// TwinCAT 3 PLC project PMS238
// ProgramVersion: 3.1.4023.0
// libraries:
//   Tc2_Math, * (Beckhoff Automation GmbH)
//   Tc2_ModbusSrv, * (Beckhoff Automation GmbH)
//   Tc2_Standard, * (Beckhoff Automation GmbH)
//   Tc2_SUPS, * (Beckhoff Automation GmbH)
//   Tc2_System, * (Beckhoff Automation GmbH)
//   Tc2_Utilities, * (Beckhoff Automation GmbH)
//   Tc3_Module, * (Beckhoff Automation GmbH)
//   Tc3_PMS_Ex, * (Beckhoff Automation GmbH)
// project tree:
//   DUTs/ AliasOnlyThisProject.TcDUT, E_CompareTime.TcDUT
//   DUTs/ION9000/ E_PM_ION9000_Address.TcDUT
//   DUTs/PM_Simulate/ E_listMeterName.TcDUT, E_PM_Simulate.TcDUT
//   Function/ CompareTime.TcPOU, FgenerateRandom.TcPOU, FUN_Compare_Timestructs.TcPOU (not stored), F_RoundLrealEx.TcPOU, IsGoodData.TcPOU, TimeStruct_To_sTimeAveva.TcPOU
//   GVLs/ GVL.TcGVL, pmDev.TcGVL
//   / PersistanceData.TcTTO, PlcTask.TcTTO
//   Persistance/ Prg_Persistance.TcPOU
//   POUs/CalAccum/ FB_CalCulateAccumulation.TcPOU
//   POUs/CrossCheckTime/ FB_TimeCrossCheck2System.TcPOU (not stored)
//   POUs/FIFO/ FB_FIFO_Lreal.TcPOU, FB_FIFO_TimeStruct.TcPOU (not stored), FB_Universal_FIFO.TcPOU, I_FIFO_Lreal.TcIO (not stored), I_FIFO_Timestruct.TcIO (not stored), I_Universal_FIFO.TcIO (not stored)
//   POUs/Metters/ FB_InitPM.TcPOU, FB_PM_ION_9000.TcPOU, FB_ReadPM5350.TcPOU, FB_READPM5500.TcPOU
//   POUs/Platform/File Logger/ FB_FileLogger.TcPOU (not stored), I_FileLogger.TcIO (not stored)
//   POUs/Platform/ PRG_MachineLogger.TcPOU
//   POUs/Program/ IP231.TcPOU, IP232.TcPOU, IP233.TcPOU, IP234.TcPOU, Ip235.TcPOU, IP236.TcPOU, IP237.TcPOU, MAIN.TcPOU, PmReport2.TcPOU
//   TEST/ FB_PmSimulate.TcPOU, PgrTest.TcPOU, PGRTestFB.TcPOU
//   Universal/DUTs/Utilities/File Logger/ E_FileLoggerAddLogsState.TcDUT (not stored), E_FileLoggerInitState.TcDUT (not stored), E_FileLoggerSetNewPathState.TcDUT (not stored), E_FileLoggerState.TcDUT (not stored)
//   Universal/Utilities/StringMerge/ FUN_MergeLongStrings10.TcPOU (not stored), FUN_MergeStrings10.TcPOU (not stored), FUN_MergeStrings3.TcPOU (not stored), FUN_MergeStrings4.TcPOU (not stored), FUN_MergeStrings5.TcPOU (not stored), FUN_MergeStrings6.TcPOU (not stored)
// real-time tasks:
//   TASK PlcTask: cycle T#10ms, priority 20, ADS port 350
//   TASK PersistanceData: cycle T#2ms, priority 2, ADS port 351

CONFIGURATION PMS238
    RESOURCE PLC ON TwinCAT3
        TASK PersistanceData(INTERVAL := T#2ms, PRIORITY := 2);
        TASK PlcTask(INTERVAL := T#10ms, PRIORITY := 20);
        PROGRAM Prg_Persistance WITH PersistanceData : Prg_Persistance;
        PROGRAM MAIN WITH PlcTask : MAIN;
        PROGRAM PRG_MachineLogger WITH PlcTask : PRG_MachineLogger;
        PROGRAM PmReport2 WITH PlcTask : PmReport2;
    END_RESOURCE
END_CONFIGURATION

// ---- DUTs/AliasOnlyThisProject.TcDUT
TYPE AliasOnlyThisProject :
STRUCT 
	systemTime : TIMESTRUCT;
	bValid : BOOL := true;
END_STRUCT
END_TYPE

// ---- DUTs/E_CompareTime.TcDUT
{attribute 'strict'}
TYPE E_CompareTime :
(
	INVALID_PRE_TIME		:= 0,
	NEW_MINUTE := 5,
	NEW_HOUR := 10,
	NEW_DAY	:= 20,
	NEW_MONTH := 30,
	NEW_YEAR	:= 32,
	SAME_MINUTE := 35,
	SAME_HOUR := 40,
	SAME_DAY := 50,
	SAME_MONTH := 60,
	SAME_YEAR  := 70
);
END_TYPE

// ---- DUTs/ION9000/E_PM_ION9000_Address.TcDUT

TYPE E_PM_ION9000_Address :
(
		
		//ION9000_E_Current_Unbalane_A :=    3012  
		//ION9000_E_Current_Unbalane_B :=    3014  
		//ION9000_E_Current_Unbalane_C :=    3016  
		ION9000_E_Current_Unbalane_Worst :=    3018,  
		//ION9000_E_Current_Unbalane_AB :=    3038  
		//ION9000_E_Current_Unbalane_BC :=    3040  
		//ION9000_E_Current_Unbalane_CA :=    3042  
		//ION9000_E_Current_Unbalane_LL_Worst :=    3044  
		//ION9000_E_Current_Unbalane_AN :=    3046  
		//ION9000_E_Current_Unbalane_BN :=    3048  
		//ION9000_E_Current_Unbalane_CN :=    3050  
		//ION9000_E_Current_Unbalane_LN_Worst:= ,
		ION9000_E_Voltage_Unbalane_LN_Worst :=    3052,  
		ION9000_E_Real_PowerA :=    3054  ,
		ION9000_E_Real_PowerB :=    3056  ,
		ION9000_E_Real_PowerC :=    3058  ,
		ION9000_E_Real_PowerTotal :=    3060  ,
		ION9000_E_Reactive_PowerA :=    3062  ,
		ION9000_E_Reactive_PowerB :=    3064  ,
		ION9000_E_Reactive_PowerC :=    3066  ,
		ION9000_E_Reactive_PowerTotal :=    3068 , 
		ION9000_E_Apparent_PowerA :=    3070  ,
		ION9000_E_Apparent_PowerB :=    3072  ,
		ION9000_E_Apparent_PowerC :=    3074  ,
		ION9000_E_Apparent_PowerTotal :=    3076  ,
		ION9000_E_Voltage_AB :=    3020 , 
		ION9000_E_Voltage_BC :=    3022  ,
		ION9000_E_Voltage_CA :=    3024  ,
		ION9000_E_Voltage_LLAvg :=    3026  ,
		ION9000_E_Voltage_AN :=    3028  ,
		ION9000_E_Voltage_BN :=    3030  ,
		ION9000_E_Voltage_CN :=    3032  ,
		ION9000_E_Voltage_NG	:= 3034,
		ION9000_E_Voltage_LNAvg :=    3036  ,
//		ION9000_E_THDF_Voltage_AB :=    22  ,
//		ION9000_E_THDF_Voltage_BC :=    24  ,
//		ION9000_E_THDF_Voltage_CA :=    26  ,
		//ION9000_E_THDF_Voltage_LL :=    28  ,
		ION9000_E_THDF_Voltage_AN :=    21330, 
		ION9000_E_THDF_Voltage_BN :=    21332, 
		ION9000_E_THDF_Voltage_CN :=    21334, 
		ION9000_E_THDF_Voltage_LN :=    21336,  
//		ION9000_E_thdR_Voltage_AB :=    40,  
//		ION9000_E_thdR_Voltage_BC :=    42,  
//		ION9000_E_thdR_Voltage_CA :=    44 , 
//		ION9000_E_thdR_Voltage_LL :=    45 , 
//		ION9000_E_thdR_Voltage_AN :=    48 , 
//		ION9000_E_thdR_Voltage_BN :=    50 , 
//		ION9000_E_thdR_Voltage_CN :=    52 , 
//		ION9000_E_thdR_Voltage_LN :=    56 , 
		ION9000_E_Current_A :=    3000 , 
		ION9000_E_Current_B :=    3002,  
		ION9000_E_Current_C :=    3004  ,
		ION9000_E_Current_N :=    3006 , 
		ION9000_E_Current_G :=    3008  ,
		ION9000_E_Current_Avg :=    3010 , 
		ION9000_E_THDF_Current_A :=    21300 , 
		ION9000_E_THDF_Current_B :=  	21302, 
		ION9000_E_THDF_Current_C :=   21304  ,
		ION9000_E_THDF_Current_N :=    21306, 
		ION9000_E_THDF_Current_G :=   21308  ,
//		ION9000_E_thdR_Current_A :=    10  ,
//		ION9000_E_thdR_Current_B :=    12  ,
//		ION9000_E_thdR_Current_C :=    14  ,
//		ION9000_E_thdR_Current_N :=    16  ,
//		ION9000_E_thdR_Current_G :=    18  ,
//		ION9000_E_Total_Demand_Distortion :=    20  
		ION9000_E_RealEnergy_IntoLoad :=    3204  ,
		ION9000_E_RealEnergy_OutLoad :=    3208 , 
		ION9000_E_RealEnergy_Absolute :=    3212  ,
		ION9000_E_RealEnergy_Signed :=    3216  ,
		ION9000_E_ReactiveEnergy_IntoLoad :=    3220 , 
		ION9000_E_ReactiveEnergy_OutLoad :=    3224  ,
		ION9000_E_ReactiveEnergy_Absolute :=    3228  ,
		ION9000_E_ReactiveEnergy_Signed :=    3232  ,
		ION9000_E_ApparentEnergy_IntoLoad :=    3236  ,
		ION9000_E_ApparentEnergy_OutLoad :=    3240  ,
		ION9000_E_ApparentEnergy :=    3244  ,
		ION9000_E_ApparentEnergy_Delivered_Received :=    3248  ,
		ION9000_E_Frequency :=    3110  ,
		ION9000_E_PowerFactor :=    3150
	
);
END_TYPE

// ---- DUTs/PM_Simulate/E_listMeterName.TcDUT
{attribute 'strict'}
TYPE E_listMeterName :
(
	LV01  := 0,
	DB_PR1_1  := 1,
	DB1  := 2,
	DB2  := 3,
	DB3  := 4,
	DB4  := 5,
	DB1_1  := 6,
	DB2_1  := 7,
	DB3_1  := 8,
	DB4_1  := 9,
	DB5  := 10,
	DB6  := 11,
	DB7  := 12,
	DB_MR  := 13,
	DB5_1  := 14,
	DB6_1  := 15,
	DB7_1  := 16,
	LV02  := 17,
	DB_PR1_2  := 18,
	DB_AIRCOMP  := 19,
	DB_AHU  := 20,
	DB8  := 21,
	DB9  := 22,
	DB10  := 23,
	DB8_1  := 24,
	DB9_1  := 25,
	DB10_1  := 26,
	A1  := 27,
	A2  := 28,
	A3  := 29,
	A4  := 30,
	A5  := 31,
	LP_PR1A  := 32,
	LP_PR1B  := 33,
	LP_PR2A  := 34,
	LP_PR2B  := 35,
	LP_PR3A  := 36,
	DB_WH  := 37,
	LP_PR3B  := 38,
	LP_PR4A  := 39,
	LP_PR4B  := 40,
	LP_BM  := 41,
	DB_BM  := 42,
	LV03  := 43,
	DB_MVAC1  := 44,
	DB_MVAC2  := 45,
	DB_OFF2  := 46,
	LP_EL1  := 47,
	LP_EL2  := 48,
	DB_OFF1  := 49,
	DB_KIT  := 50,
	LP_WH2  := 51,
	LP_WH1  := 52,
	CH4  := 53,
	CH5  := 54,
	CH6  := 55,
	LV04  := 56,
	DB_PR2  := 57,
	DB11  := 58,
	DB12  := 59,
	DB13  := 60,
	DB14  := 61,
	DB11_1  := 62,
	DB12_1  := 63,
	DB13_1  := 64,
	DB14_1  := 65,
	DB15  := 66,
	DB15_1  := 67,
	LP_PR5A  := 68,
	LP_PR5B  := 69,
	LP_PR6A  := 70,
	LP_PR6B  := 71,
	 DB1_2	 :=72,
	 DB2_2	 :=73,
	 DB3_2	 :=74,
	 DB4_2	 :=75,
	 DB5_2	 :=76,
	 DB6_2	 :=77,
	 DB7_2	 :=78,
	 DB8_2	 :=79,
	 DB9_2	 :=80,
	 DB10_2	 :=81,
	 DB11_2	 :=82,
	 DB12_2	 :=83,
	 DB13_2	 :=84,
	 DB14_2	 :=85,
	 DB15_2	 :=86
);
END_TYPE

// ---- DUTs/PM_Simulate/E_PM_Simulate.TcDUT

{attribute 'strict'}
TYPE E_PM_Simulate :
(
	
	PM_SIMU_WAIT := 0,
	PM_SIMU_UPDATE := 10,
	PM_SIMU_READ_FAULT := 20
);
END_TYPE

// ---- GVLs/GVL.TcGVL

VAR_GLOBAL
	fbMachineLogger : FB_FileLogger;
	fbMachineTime	: AliasOnlyThisProject;
END_VAR
VAR_GLOBAL CONSTANT
	TIME_INIT	: TIME := T#30S;
END_VAR

// ---- GVLs/pmDev.TcGVL
{attribute 'qualified_only'}
VAR_GLOBAL
	DB01_02_5350		: ST_PowerMeter; //DB12.1
	DB01_03_5350		: ST_PowerMeter; //DB11.1
	DB01_05_5350		: ST_PowerMeter; //LP-PR6B
	DB01_06_5350		: ST_PowerMeter; //LP-PR6A
	DB01_12_5350		: ST_PowerMeter; //LP-WH2
	
	DB01_01_5500		: ST_PowerMeter; //DB12
	DB01_04_5500		: ST_PowerMeter; //DB11
	DB01_07_5500		: ST_PowerMeter; //DB-PR2
	DB01_11_5500		: ST_PowerMeter; //LP-WH1
	DB01_18_5500		: ST_PowerMeter; //DB-WH
	DB01_20_5500		: ST_PowerMeter; //LP-BM
	DB01_22_5500		: ST_PowerMeter; //DB-BM 
	
	DB02_01_5350		: ST_PowerMeter; //DB13.1
	DB02_03_5350		: ST_PowerMeter; //DB15.1
	DB02_05_5350		: ST_PowerMeter; //DB14.1 
	DB02_07_5350		: ST_PowerMeter; //LP-PR5B
	DB02_08_5350		: ST_PowerMeter; //LP-PR5A
	
	DB02_02_5500		: ST_PowerMeter; //DB13
	DB02_04_5500		: ST_PowerMeter; //DB15
	DB02_06_5500		: ST_PowerMeter; //DB14
	
	
	DB03_01_5350		: ST_PowerMeter; //DB7.1
	DB03_03_5350		: ST_PowerMeter; //DB5.1 
	DB03_05_5350		: ST_PowerMeter; //DB6.1
	DB03_07_5350		: ST_PowerMeter; //LP-PR3B
	DB03_08_5350		: ST_PowerMeter; //LP-PR3A
	
	DB03_02_5500		: ST_PowerMeter; //DB7
	DB03_04_5500		: ST_PowerMeter; //DB5
	DB03_06_5500		: ST_PowerMeter; //DB6
	
	DB04_01_5350		: ST_PowerMeter; //DB4.1 
	DB04_03_5350		: ST_PowerMeter; //DB3.1 
	DB04_05_5350		: ST_PowerMeter; //DB2.1 
	DB04_07_5350		: ST_PowerMeter; //LP-PR4B
	DB04_08_5350		: ST_PowerMeter; //LP-PR4A
	
	DB04_02_5500		: ST_PowerMeter; //DB4
	DB04_04_5500		: ST_PowerMeter; //DB3
	DB04_06_5500		: ST_PowerMeter; //DB2
	
	
	DB05_01_5350		: ST_PowerMeter; //LP-PR1A
	DB05_02_5350		: ST_PowerMeter; //LP-PR1B
	DB05_03_5350		: ST_PowerMeter; //DB8.1 
	DB05_05_5350		: ST_PowerMeter; //DB9.1 
	DB05_07_5350		: ST_PowerMeter; //DB10.1
	DB05_09_5350		: ST_PowerMeter; //DB1.1
	DB05_21_5350		: ST_PowerMeter; //LP-PR2B
	DB05_22_5350		: ST_PowerMeter; //LP-PR2A
	
	DB05_04_5500		: ST_PowerMeter; //DB8
	DB05_06_5500		: ST_PowerMeter; //DB9
	DB05_08_5500		: ST_PowerMeter; //DB10
	DB05_10_5500		: ST_PowerMeter; //DB1 
	
	DB06_01_5500		: ST_PowerMeter; //LP-EL2
	DB06_02_5500		: ST_PowerMeter; //LV-SECTION4
	DB06_03_5500		: ST_PowerMeter; //LP-EL1
	DB06_04_5500		: ST_PowerMeter; //LV-SECTION3
	DB06_05_5500		: ST_PowerMeter; //DB-PR1 (S2) 
	DB06_06_5500		: ST_PowerMeter; //DB-PR1(S1)
	DB06_07_5500		: ST_PowerMeter; //DB-AHU
	DB06_08_5500		: ST_PowerMeter; //DB-OFF1
	DB06_11_5500		: ST_PowerMeter; //DB-MR
	DB06_33_5500		: ST_PowerMeter; //DB-KIT
	DB06_38_5500		: ST_PowerMeter; //DB-OFF2
	
	DB07_01_5500		: ST_PowerMeter; //LV-SECTION1
	DB07_02_5500		: ST_PowerMeter; // LV-SECTION2
	DB07_03_5500		: ST_PowerMeter; //DB-AIRCOMP 
	DB07_04_5500		: ST_PowerMeter; //DB-MVAC2
	DB07_05_5500		: ST_PowerMeter; //DB-MVAC1
	///////////////////////////////////////////////Sun update Code
	DB07_06_5350		: ST_PowerMeter; // A1
	DB07_07_5350		: ST_PowerMeter; //A2
	DB07_08_5350		: ST_PowerMeter; //A3
	DB07_09_5350		: ST_PowerMeter; //A4
	DB07_10_5350		: ST_PowerMeter; //A5
	DB07_11_5350		: ST_PowerMeter; //CH4
	DB07_12_5350		: ST_PowerMeter; //CH5
	DB07_13_5350		: ST_PowerMeter; //CH6
	/////// virtual metter 
	PowerMeter_Db1_2	: st_powerMeter;// DB1.2
	PowerMeter_Db2_2	: ST_PowerMeter;
	PowerMeter_db3_2	: ST_PowerMeter;
	PowerMeter_db4_2	: ST_PowerMeter;
	PowerMeter_db5_2	: ST_PowerMeter;
	powerMeter_db6_2	: ST_PowerMeter;
	PowerMeter_db7_2	: ST_PowerMeter;
	PowerMeter_db8_2	: ST_PowerMeter;
	PowerMeter_db9_2	: ST_PowerMeter;
	PowerMeter_db10_2	: ST_PowerMeter;
	PowerMeter_db11_2	: ST_PowerMeter;
	PowerMeter_db12_2	: ST_PowerMeter;
	PowerMeter_db13_2	: ST_PowerMeter;
	PowerMeter_db14_2	: ST_PowerMeter;
	PowerMeter_db15_2	: ST_PowerMeter;

	// new meter
	PowerMeter_Lv01		: ST_PowerMeter;
	PowerMeter_Lv02		: ST_PowerMeter;
	PowerMeter_Lv03		: ST_PowerMeter;
	PowerMeter_Lv04		: ST_PowerMeter;

	NT_GetTime : NT_GetTime;
	AvevaTimeStruct : TIMESTRUCT;
	bAlarmDifferentTime2System : BOOL;
END_VAR
VAR_GLOBAL CONSTANT
	TIMESTRUCT_DEFAULT : TIMESTRUCT;
	InvalidValueEnergyIntoload   : LREAL := 1E12; // if Energy Intoload bigger this parameter or lower than (-NanEnergyIntoload) , EnergyIntoload can't be use
	numAllMeter	 :UINT := 87;
	SecondDifferentAllow : UDINT := 300;
END_VAR
// commissioning
VAR_GLOBAL
	bTrigReadCOmmision : BOOL;
END_VAR

// ---- Persistance/Prg_Persistance.TcPOU
PROGRAM Prg_Persistance
VAR
FB_S_UPS_CX8190	: FB_S_UPS_CX81xx;

END_VAR

FB_S_UPS_CX8190(	sNetID :='',
					iPLCPort        := 851, (* PLC Runtime System for writing persistent data *)
  					tTimeout        := DEFAULT_ADS_TIMEOUT, (* ADS Timeout *)
    				eUpsMode        := eSUPS_WrPersistData_Shutdown, (* UPS mode (w/wo writing persistent data, w/wo NO shutdown) *)
   					ePersistentMode := SPDM_2PASS, (* mode for writing persistent data *)
    				tRecoverTime    := T#10S, (* ON time to recover from short power failure in mode eSUPS_WrPersistData_NoShutdown/eSUPS_CheckPowerStatus *)
					);

END_PROGRAM

// ---- POUs/Program/MAIN.TcPOU
PROGRAM MAIN
VAR
	fb_timeCrossCheck	: FB_TimeCrossCheck2System;
	eEgxRead	: UINT := WAIT_EGX_FREE;
END_VAR

VAR CONSTANT
	WAIT_EGX_FREE	: UINT := 0;
	EGX_231 : UINT := 231;
	EGX_232 : UINT := 232;
	EGX_233 : UINT := 233;
	EGX_234 : UINT := 234;
	EGX_235 : UINT := 235;
	EGX_236 : UINT := 236;
	EGX_237 : UINT := 237;
END_VAR

IF FUN_Compare_Timestructs(
	ts1 := pmDev.AvevaTimeStruct, 
	ts2 := pmDev.TIMESTRUCT_DEFAULT
	) = 0 // equal
THEN
	 pmDev.bAlarmDifferentTime2System := FALSE;
	 
ELSE 
	fb_timeCrossCheck(	TimeStruct_Sys1 := pmDev.AvevaTimeStruct,
					TimeStruct_Sys2 := pmDev.NT_GetTime.TIMESTR,
					secondDifferentAllow := pmdev.SecondDifferentAllow,
					bErrorTimeTwoSystem => pmDev.bAlarmDifferentTime2System);
END_IF

pmdev.NT_GetTime(START := FALSE);
pmdev.NT_GetTime(
	START := TRUE,
	TIMESTR => GVL.fbMachineTime.systemTime
); 
					
IP231();
IP232();
IP233();
IP234();
IP235();
IP236();
IP237();
CASE eEgxRead OF
	WAIT_EGX_FREE :
		IF NOT IP231.Busy
		AND NOT IP232.Busy
		AND NOT IP233.Busy
		AND NOT IP234.Busy
		AND NOT IP235.Busy
		AND NOT IP236.Busy
		AND NOT IP237.Busy
		THEN
			eEgxRead := EGX_231;
		END_IF
		
	EGX_231 :
		IP231.Mr_Read();
		IF NOT IP231.Busy THEN
			eEgxRead := EGX_232;
		END_IF
		
	EGX_232 :
		IP232.Mr_Read();
		IF NOT IP232.Busy THEN
			eEgxRead := EGX_233;
		END_IF
		
	EGX_233 :
		IP233.Mr_Read();
		IF NOT IP233.Busy THEN
			eEgxRead := EGX_234;
		END_IF
		
	EGX_234 :
		IP234.Mr_Read();
		IF NOT IP234.Busy THEN
			eEgxRead := EGX_235;
		END_IF
		
	EGX_235 :
		IP235.Mr_Read();
		IF NOT IP235.Busy THEN
			eEgxRead := EGX_236;
		END_IF
		
	EGX_236 :
		IP236.Mr_Read();
		IF NOT IP236.Busy THEN
			eEgxRead := EGX_237;
		END_IF
		
	EGX_237 :
		IP237.Mr_Read();
		IF NOT IP237.Busy THEN
			eEgxRead := WAIT_EGX_FREE;
		END_IF
END_CASE

pmdev.bTrigReadCOmmision := FALSE;
CalculateVirtualMeter(	MeterMain := pmDev.DB05_10_5500 ,
						MeterSub := pmDev.DB05_09_5350,
						MeterVirtual := pmDev.PowerMeter_Db1_2);
						
 CalculateVirtualMeter( MeterMain := pmDev.DB04_06_5500,
                      MeterSub := pmDev.DB04_05_5350,
                       MeterVirtual :=  pmDev.PowerMeter_Db2_2);
 
 CalculateVirtualMeter( MeterMain := pmDev.DB04_04_5500,
                      MeterSub :=  pmDev.DB04_03_5350,
                       MeterVirtual :=  pmDev.PowerMeter_db3_2);
 
 CalculateVirtualMeter( MeterMain := pmDev.DB04_02_5500,
                      MeterSub := pmDev.DB04_01_5350,
                       MeterVirtual :=  pmDev.PowerMeter_db4_2);
 
 CalculateVirtualMeter( MeterMain := pmDev.DB03_04_5500,
                      MeterSub := pmDev.DB03_03_5350,
                       MeterVirtual :=  pmDev.PowerMeter_db5_2);
 
 CalculateVirtualMeter( MeterMain := pmDev.DB03_06_5500,
                      MeterSub := pmDev.DB03_05_5350,
                       MeterVirtual :=  pmDev.powerMeter_db6_2);
 
 CalculateVirtualMeter( MeterMain := pmDev.DB03_02_5500,
                      MeterSub := pmDev.DB03_01_5350,
                       MeterVirtual :=  pmDev.PowerMeter_db7_2);
 
 CalculateVirtualMeter( MeterMain := pmDev.DB05_04_5500,
                      MeterSub := pmDev.DB05_03_5350,
                       MeterVirtual :=  pmDev.PowerMeter_db8_2);
 
 CalculateVirtualMeter( MeterMain := pmDev.DB05_06_5500,
                      MeterSub := pmDev.DB05_05_5350,
                       MeterVirtual :=  pmDev.PowerMeter_db9_2);
 
 CalculateVirtualMeter( MeterMain := pmDev.DB05_08_5500,
                      MeterSub := pmDev.DB05_07_5350,
                       MeterVirtual :=  pmDev.PowerMeter_db10_2);
 
 CalculateVirtualMeter( MeterMain := pmDev.DB01_04_5500,
                      MeterSub := pmDev.DB01_03_5350,
                       MeterVirtual :=  pmDev.PowerMeter_db11_2);
 
 CalculateVirtualMeter( MeterMain :=  pmDev.DB01_01_5500,
                      MeterSub := pmDev.DB01_02_5350,
                       MeterVirtual :=  pmDev.PowerMeter_db12_2);
 
 CalculateVirtualMeter( MeterMain := pmDev.DB02_02_5500,
                      MeterSub := pmDev.DB02_01_5350,
                       MeterVirtual :=  pmDev.PowerMeter_db13_2);
 
 CalculateVirtualMeter( MeterMain := pmDev.DB02_06_5500,
                      MeterSub := pmDev.DB02_05_5350,
                       MeterVirtual :=  pmDev.PowerMeter_db14_2);
 
 CalculateVirtualMeter( MeterMain := pmDev.DB02_04_5500,
                      MeterSub := pmDev.DB02_03_5350,
                       MeterVirtual :=  pmDev.PowerMeter_db15_2);

METHOD CalculateVirtualMeter : BOOL
VAR_INPUT
	MeterMain	: REFERENCE TO  ST_PowerMeter;// meterVirtual := MeterMain - MeterSub
	MeterSub	: REFERENCE TO ST_PowerMeter;// meterVirtual := MeterMain - MeterSub
	MeterVirtual : REFERENCE TO ST_PowerMeter; // meterVirtual := MeterMain - MeterSub
END_VAR
VAR_OUTPUT
	
END_VAR
	MeterVirtual.Basic.Current_Avg := MeterMain.Basic.Current_Avg - MeterSub.Basic.Current_Avg;
	MeterVirtual.Basic.Real_PowerTotal := MeterMain.Basic.Real_PowerTotal - MeterSub.Basic.Real_PowerTotal;
	MeterVirtual.Basic.RealEnergy_IntoLoad  := MeterMain.Basic.RealEnergy_IntoLoad - MeterSub.Basic.RealEnergy_IntoLoad;
END_METHOD

END_PROGRAM

// ---- POUs/Program/IP231.TcPOU
PROGRAM IP231
VAR
	timer				: TON;
	nState				: INT := STATE_INIT;
	
	fbInit231_02_5350			: FB_InitPM;
	fbInit231_03_5350			: FB_InitPM;
	fbInit231_05_5350			: FB_InitPM;
	fbInit231_06_5350			: FB_InitPM;
	fbInit231_12_5350			: FB_InitPM;
	
	fbRead231_02_5350			: FB_ReadPM5350;
	fbRead231_03_5350			: FB_ReadPM5350;
	fbRead231_05_5350			: FB_ReadPM5350;
	fbRead231_06_5350			: FB_ReadPM5350;
	fbRead231_12_5350			: FB_ReadPM5350;
	
	fbInit231_01_5500			: FB_InitPM;
	fbInit231_04_5500			: FB_InitPM;
	fbInit231_07_5500			: FB_InitPM;
	fbInit231_11_5500			: FB_InitPM;
	fbInit231_18_5500			: FB_InitPM;
	fbInit231_20_5500			: FB_InitPM;
	fbInit231_22_5500			: FB_InitPM;
	
	fbRead231_01_5500			: FB_ReadPM5500;
	fbRead231_04_5500			: FB_ReadPM5500;
	fbRead231_07_5500			: FB_ReadPM5500;
	
	//Update 29-8-2022
	fbRead231_11_5500			: FB_ReadPM5350;
	
	fbRead231_18_5500			: FB_ReadPM5500;
	fbRead231_20_5500			: FB_ReadPM5500;
	fbRead231_22_5500			: FB_ReadPM5500;
END_VAR

VAR CONSTANT
	STATE_INIT			:	INT		:= 0;
	STATE_WAIT_CMD		: 	INT		:= 5;
	STATE_READ2			:	INT		:= 20;
	STATE_READ3			:	INT		:= 30;
	STATE_READ5			:	INT		:= 50;
	STATE_READ6			:	INT		:= 60;
	STATE_READ12		:	INT		:= 90;
	STATE_READ1			:	INT		:= 10;
	STATE_READ4			:	INT		:= 40;
	STATE_READ7			:	INT		:= 70;
	STATE_READ11		:	INT		:= 110;
	STATE_READ18		:	INT		:= 180;
	STATE_READ20		:	INT		:= 200;
	STATE_READ22		:	INT		:= 220;
END_VAR

CASE nState OF
	STATE_INIT:
		fbInit231_02_5350(	sIpAddress	:= '10.91.37.231',
							nPort		:= 502,
							nUnitID		:= 2,
							PM			:= pmDev.DB01_02_5350);
		fbInit231_03_5350(	sIpAddress	:= '10.91.37.231',
							nPort		:= 502,
							nUnitID		:= 03,
							PM			:= pmDev.DB01_03_5350);
		fbInit231_05_5350(	sIpAddress	:= '10.91.37.231',
							nPort		:= 502,
							nUnitID		:= 5,
							PM			:= pmDev.DB01_05_5350);
		fbInit231_06_5350(	sIpAddress	:= '10.91.37.231',
							nPort		:= 502,
							nUnitID		:= 6,
							PM			:= pmDev.DB01_06_5350);
							
		fbInit231_11_5500(	sIpAddress	:= '10.91.37.231',
							nPort		:= 502,
							nUnitID		:= 11,
							PM			:= pmDev.DB01_11_5500);
							
		fbInit231_12_5350(	sIpAddress	:= '10.91.37.231',
							nPort		:= 502,
							nUnitID		:= 12,
							PM			:= pmDev.DB01_12_5350);
							
		fbInit231_01_5500(	sIpAddress	:= '10.91.37.231',
							nPort		:= 502,
							nUnitID		:= 1,
							PM			:= pmDev.DB01_01_5500);
		fbInit231_04_5500(	sIpAddress	:= '10.91.37.231',
							nPort		:= 502,
							nUnitID		:= 4,
							PM			:= pmDev.DB01_04_5500);
		fbInit231_07_5500(	sIpAddress	:= '10.91.37.231',
							nPort		:= 502,
							nUnitID		:= 7,
							PM			:= pmDev.DB01_07_5500);
		
		fbInit231_18_5500(	sIpAddress	:= '10.91.37.231',
							nPort		:= 502,
							nUnitID		:= 18,
							PM			:= pmDev.DB01_18_5500);
		fbInit231_20_5500(	sIpAddress	:= '10.91.37.231',
							nPort		:= 502,
							nUnitID		:= 20,
							PM			:= pmDev.DB01_20_5500);
		fbInit231_22_5500(	sIpAddress	:= '10.91.37.231',
							nPort		:= 502,
							nUnitID		:= 22,
							PM			:= pmDev.DB01_22_5500);
							
		timer(In:=TRUE, PT:= TIME_INIT);
		IF timer.Q THEN
			timer(In := FALSE);
			nState	:= STATE_WAIT_CMD;
		END_IF
	STATE_WAIT_CMD:
		;
	STATE_READ2:
		fbRead231_02_5350(
			bExecute:=TRUE,
			PM:= pmDev.DB01_02_5350);
		IF NOT fbRead231_02_5350.Q THEN
			nState	:= STATE_READ3;
			fbRead231_02_5350(
				bExecute:=FALSE,
				PM:= pmDev.DB01_02_5350);
		END_IF
		
	STATE_READ3:
		fbRead231_03_5350(
			bExecute:=TRUE,
			PM:= pmDev.DB01_03_5350);
		IF NOT fbRead231_03_5350.Q THEN
			nState	:= STATE_READ5;
			fbRead231_03_5350(
				bExecute:=FALSE,
				PM:= pmDev.DB01_03_5350);
		END_IF	
	
	STATE_READ5:
		fbRead231_05_5350(
			bExecute:=TRUE,
			PM:= pmDev.DB01_05_5350);
		IF NOT fbRead231_05_5350.Q THEN
			nState	:= STATE_READ6;
			fbRead231_05_5350(
				bExecute:=FALSE,
				PM:= pmDev.DB01_05_5350);
		END_IF	
		
	STATE_READ6:
		fbRead231_06_5350(
			bExecute:=TRUE,
			PM:= pmDev.DB01_06_5350);
		IF NOT fbRead231_06_5350.Q THEN
			nState	:= STATE_READ11;
			fbRead231_06_5350(
			bExecute:=FALSE,
			PM := pmDev.DB01_06_5350);
		END_IF
		
	STATE_READ11:
	
		
		fbRead231_11_5500(
			bExecute:=TRUE,
			PM:= pmDev.DB01_11_5500);
		IF NOT fbRead231_11_5500.Q THEN
			nState	:= STATE_READ12;
			fbRead231_11_5500(
				bExecute:=FALSE,
				PM:= pmDev.DB01_11_5500);
		END_IF
		
	STATE_READ12:
		fbRead231_12_5350(
			bExecute:=TRUE,
			PM:= pmDev.DB01_12_5350);
		IF NOT fbRead231_12_5350.Q THEN
			nState	:= STATE_READ1;
			fbRead231_12_5350(
				bExecute:=FALSE,
				PM:= pmDev.DB01_12_5350);
		END_IF	
	STATE_READ1:
		fbRead231_01_5500(
			bExecute:=TRUE,
			PM:= pmDev.DB01_01_5500);
		IF NOT fbRead231_01_5500.Q THEN
			nState	:= STATE_READ4;
			fbRead231_01_5500(
				bExecute:=FALSE,
				PM:= pmDev.DB01_01_5500);
		END_IF
	STATE_READ4:
		fbRead231_04_5500(
			bExecute:=TRUE,
			PM:= pmDev.DB01_04_5500);
		IF NOT fbRead231_04_5500.Q THEN
			nState	:= STATE_READ7;
			fbRead231_04_5500(
				bExecute:=FALSE,
				PM:= pmDev.DB01_04_5500);
		END_IF
	
	STATE_READ7:
		fbRead231_07_5500(
			bExecute:=TRUE,
			PM:= pmDev.DB01_07_5500);
		IF NOT fbRead231_07_5500.Q THEN
			nState	:= STATE_READ18;
			fbRead231_07_5500(
				bExecute:=FALSE,
				PM:= pmDev.DB01_07_5500);
		END_IF
		
	STATE_READ18:
		fbRead231_18_5500(
			bExecute:=TRUE,
			PM:= pmDev.DB01_18_5500);
		IF NOT fbRead231_18_5500.Q THEN
			nState	:= STATE_READ20;
			fbRead231_18_5500(
				bExecute:=FALSE,
				PM:= pmDev.DB01_18_5500);
		END_IF
		
	STATE_READ20:
		fbRead231_20_5500(
			bExecute:=TRUE,
			PM:= pmDev.DB01_20_5500);
		IF NOT fbRead231_20_5500.Q THEN
			nState	:= STATE_READ22;
			fbRead231_20_5500(
				bExecute:=FALSE,
				PM:= pmDev.DB01_20_5500);
		END_IF
	
	STATE_READ22:
		fbRead231_22_5500(
			bExecute:=TRUE,
			PM:= pmDev.DB01_22_5500);
		IF NOT fbRead231_22_5500.Q THEN
			nState	:= STATE_WAIT_CMD;
			fbRead231_22_5500(
				bExecute:=FALSE,
				PM:= pmDev.DB01_22_5500);
		END_IF
	
END_CASE

PROPERTY Busy : Bool
GET
Busy := nState <> STATE_WAIT_CMD;
END_GET
END_PROPERTY

METHOD Mr_Read : BOOL
VAR_INPUT
END_VAR
IF nState = STATE_WAIT_CMD THEN
	nState := STATE_READ2;
END_IF
END_METHOD

END_PROGRAM

// ---- POUs/Metters/FB_InitPM.TcPOU
FUNCTION_BLOCK FB_InitPM
VAR_INPUT
	sIpAddress		: STRING;
	nUnitID			: BYTE;
	nPort			: UINT;
END_VAR

VAR_OUTPUT
END_VAR

VAR_IN_OUT
	PM		:	ST_PowerMeter;
END_VAR

VAR
END_VAR

(******** Init Connection **************)
PM.Conn.sIPAddress		:= sIpAddress;
PM.Conn.nUnitID			:= nUnitID;
PM.Conn.nPort			:= nPort;

END_FUNCTION_BLOCK

// ---- POUs/Metters/FB_ReadPM5350.TcPOU
FUNCTION_BLOCK FB_ReadPM5350 EXTENDS ReadPm5350

VAR_OUTPUT
END_VAR
VAR PERSISTENT
	validEnvergyIntoLoad : LREAL;
END_VAR
(*VAR_IN_OUT
	PM		:	ST_PowerMeter;
END_VAR*)
VAR
	bOtherDataGood : BOOL;
END_VAR

SUPER^(PM:= THIS^.PM,
		bExecute := bExecute);

bOtherdataGood := 	IsGoodData( pm.Basic.Voltage_LLAvg )
				AND IsGoodData( pm.Basic.Current_Avg)
				AND IsGoodData(	pm.Basic.Frequency)
				AND IsGoodData( pm.Basic.Voltage_AN)
				AND IsGoodData(	pm.Basic.Voltage_AB)
				AND IsGoodData( pm.Basic.Voltage_BN)
				AND IsGoodData(	pm.Basic.Voltage_BC)
				AND IsGoodData( pm.Basic.Voltage_CN)
				AND IsGoodData(	pm.Basic.Voltage_CA);
				
				
IF IsGoodData (pm.Basic.RealEnergy_IntoLoad ) AND bOtherDataGood THEN
	;// pm.Basic.RealEnergy_IntoLoad still it
	validEnvergyIntoLoad := pm.Basic.RealEnergy_IntoLoad;
ELSE
	pm.Basic.RealEnergy_IntoLoad := validEnvergyIntoLoad;
END_IF

//round value
	(*PM.Basic.RealEnergy_IntoLoad := F_RoundLrealEx(	lrIn 	:= PM.Basic.RealEnergy_IntoLoad,
										iPrecision 	:= 0);*)
												
	PM.Basic.PowerFactor := F_RoundLrealEx(	lrIn 	:= PM.Basic.PowerFactor,
								iPrecision 	:= 2);

END_FUNCTION_BLOCK

// ---- Function/IsGoodData.TcPOU
FUNCTION IsGoodData : BOOL// check into load data not nan and too big or too low
VAR_INPUT
	dataLr : LREAL;
END_VAR
VAR
END_VAR

IF LrealIsNaN( dataLr ) THEN
	IsGoodData := FALSE;
ELSIF dataLr > pmDev.InvalidValueEnergyIntoload OR dataLr <  0.0001 THEN
	IsGoodData := FALSE;
ELSE
	IsGoodData := True;
END_IF

END_FUNCTION

// ---- Function/F_RoundLrealEx.TcPOU
FUNCTION F_RoundLrealEx : LREAL
VAR_INPUT
	lrIn : LREAL;
	iPrecision : UINT;
END_VAR
VAR
	lrTemp	: LREAL;
END_VAR

lrTemp := lrIn * EXPT(10,iPrecision);
lrTemp := LTRUNC(lrTemp);
F_RoundLrealEx := lrTemp / EXPT(10,iPrecision);

END_FUNCTION

// ---- POUs/Metters/FB_READPM5500.TcPOU
FUNCTION_BLOCK FB_READPM5500 EXTENDS ReadPm5500

VAR_OUTPUT
END_VAR
VAR PERSISTENT 
	validEnvergyIntoLoad : LREAL;
END_VAR
(*VAR_IN_OUT
	PM		:	ST_PowerMeter;
END_VAR*)
VAR
	bOtherDataGood : BOOL;
END_VAR

SUPER^(PM:= THIS^.PM,
		bExecute := bExecute);

bOtherdataGood := 	IsGoodData( pm.Basic.Voltage_LLAvg )
				AND IsGoodData ( pm.Basic.Current_Avg)
				AND IsGoodData(	pm.Basic.Frequency)
				AND IsGoodData( pm.Basic.Voltage_AN)
				AND IsGoodData(	pm.Basic.Voltage_AB)
				AND IsGoodData( pm.Basic.Voltage_BN)
				AND IsGoodData(	pm.Basic.Voltage_BC)
				AND IsGoodData( pm.Basic.Voltage_CN)
				AND IsGoodData(	pm.Basic.Voltage_CA);

				
IF IsGoodData (pm.Basic.RealEnergy_IntoLoad ) AND bOtherDataGood THEN
	;// pm.Basic.RealEnergy_IntoLoad still it
	validEnvergyIntoLoad := pm.Basic.RealEnergy_IntoLoad;
ELSE
	pm.Basic.RealEnergy_IntoLoad := validEnvergyIntoLoad;
END_IF

//round value
	(*PM.Basic.RealEnergy_IntoLoad := F_RoundLrealEx(	lrIn 	:= PM.Basic.RealEnergy_IntoLoad,
										iPrecision 	:= 0);*)
												
	PM.Basic.PowerFactor := F_RoundLrealEx(	lrIn 	:= PM.Basic.PowerFactor,
								iPrecision 	:= 2);

END_FUNCTION_BLOCK

// ---- POUs/Program/IP232.TcPOU
PROGRAM IP232
VAR
	timer				: TON;	
	nState				: INT := STATE_INIT;
	
	fbInit232_01_5350			: FB_InitPM;
	fbInit232_03_5350			: FB_InitPM;
	fbInit232_05_5350			: FB_InitPM;
	fbInit232_07_5350			: FB_InitPM;
	fbInit232_08_5350			: FB_InitPM;
	
	fbRead232_01_5350			: FB_ReadPM5350;
	fbRead232_03_5350			: FB_ReadPM5350;
	fbRead232_05_5350			: FB_ReadPM5350;
	fbRead232_07_5350			: FB_ReadPM5350;
	fbRead232_08_5350			: FB_ReadPM5350;
	
	fbInit232_02_5500			: FB_InitPM;
	fbInit232_04_5500			: FB_InitPM;
	fbInit232_06_5500			: FB_InitPM;
	
	fbRead232_02_5500			: FB_ReadPM5500;
	fbRead232_04_5500			: FB_ReadPM5500;
	fbRead232_06_5500			: FB_ReadPM5500;
	
END_VAR

VAR CONSTANT
	STATE_INIT			:	INT		:= 0;
	STATE_WAIT_CMD		: 	INT		:= 5;
	STATE_READ1			:	INT		:= 10;
	STATE_READ3			:	INT		:= 30;
	STATE_READ5			:	INT		:= 50;
	STATE_READ7			:	INT		:= 70;
	STATE_READ8			:	INT		:= 80;
	STATE_READ2			:	INT		:= 20;
	STATE_READ4			:	INT		:= 40;
	STATE_READ6			:	INT		:= 60;
END_VAR

CASE nState OF
	STATE_INIT:
		fbInit232_01_5350(	sIpAddress	:= '10.91.37.232',
							nPort		:= 502,
							nUnitID		:= 1,
							PM			:= pmDev.DB02_01_5350);
		fbInit232_03_5350(	sIpAddress	:= '10.91.37.232',
							nPort		:= 502,
							nUnitID		:= 3,
							PM			:= pmDev.DB02_03_5350);
		fbInit232_05_5350(	sIpAddress	:= '10.91.37.232',
							nPort		:= 502,
							nUnitID		:= 5,
							PM			:= pmDev.DB02_05_5350);
		fbInit232_07_5350(	sIpAddress	:= '10.91.37.232',
							nPort		:= 502,
							nUnitID		:= 7,
							PM			:= pmDev.DB02_07_5350);
		fbInit232_08_5350(	sIpAddress	:= '10.91.37.232',
							nPort		:= 502,
							nUnitID		:= 8,
							PM			:= pmDev.DB02_08_5350);			
		fbInit232_02_5500(	sIpAddress	:= '10.91.37.232',
							nPort		:= 502,
							nUnitID		:= 2,
							PM			:= pmDev.DB02_02_5500);
		fbInit232_04_5500(	sIpAddress	:= '10.91.37.232',
							nPort		:= 502,
							nUnitID		:= 4,
							PM			:= pmDev.DB02_04_5500);
		fbInit232_06_5500(	sIpAddress	:= '10.91.37.232',
							nPort		:= 502,
							nUnitID		:= 6,
							PM			:= pmDev.DB02_06_5500);
							
		timer(In:=TRUE, PT:= TIME_INIT);
		IF timer.Q THEN
			timer(In:=FALSE);
			nState	:= STATE_WAIT_CMD;
		END_IF
		
	STATE_WAIT_CMD:
			;
						
	STATE_READ1:
		fbRead232_01_5350(
			bExecute:=TRUE,
			PM:= pmDev.DB02_01_5350);
		IF NOT fbRead232_01_5350.Q THEN
			nState	:= STATE_READ3;
			fbRead232_01_5350(
				bExecute:=FALSE,
				PM:= pmDev.DB02_01_5350);
		END_IF
		
	STATE_READ3:
		fbRead232_03_5350(
			bExecute:=TRUE,
			PM:= pmDev.DB02_03_5350);
		IF NOT fbRead232_03_5350.Q THEN
			nState	:= STATE_READ5;
			fbRead232_03_5350(
				bExecute:=FALSE,
				PM:= pmDev.DB02_03_5350);
		END_IF	
	
	STATE_READ5:
		fbRead232_05_5350(
			bExecute:=TRUE,
			PM:= pmDev.DB02_05_5350);
		IF NOT fbRead232_05_5350.Q THEN
			nState	:= STATE_READ7;
			fbRead232_05_5350(
				bExecute:=FALSE,
				PM:= pmDev.DB02_05_5350);
		END_IF	
		
	STATE_READ7:
		fbRead232_07_5350(
			bExecute:=TRUE,
			PM:= pmDev.DB02_07_5350);
		IF NOT fbRead232_07_5350.Q THEN
			nState	:= STATE_READ8;
			fbRead232_07_5350(
				bExecute:=FALSE,
				PM:= pmDev.DB02_07_5350);
		END_IF	
		
	STATE_READ8:
		fbRead232_08_5350(
			bExecute:=TRUE,
			PM:= pmDev.DB02_08_5350);
		IF NOT fbRead232_08_5350.Q THEN
			nState	:= STATE_READ2;
			fbRead232_08_5350(
				bExecute:=FALSE,
				PM:= pmDev.DB02_08_5350);
		END_IF	
		
	STATE_READ2:
		fbRead232_02_5500(
			bExecute:=TRUE,
			PM:= pmDev.DB02_02_5500);
		IF NOT fbRead232_02_5500.Q THEN
			nState	:= STATE_READ4;
			fbRead232_02_5500(
				bExecute:=FALSE,
				PM:= pmDev.DB02_02_5500);
		END_IF
	STATE_READ4:
		fbRead232_04_5500(
			bExecute:=TRUE,
			PM:= pmDev.DB02_04_5500);
		IF NOT fbRead232_04_5500.Q THEN
			nState	:= STATE_READ6;
			fbRead232_04_5500(
				bExecute:=FALSE,
				PM:= pmDev.DB02_04_5500);
		END_IF
	
	STATE_READ6:
		fbRead232_06_5500(
			bExecute:=TRUE,
			PM:= pmDev.DB02_06_5500);
		IF NOT fbRead232_06_5500.Q THEN
			nState	:= STATE_WAIT_CMD;
			fbRead232_06_5500(
				bExecute:=FALSE,
				PM:= pmDev.DB02_06_5500);
		END_IF
		
END_CASE

PROPERTY Busy : Bool
GET
Busy := nState <> STATE_WAIT_CMD;
END_GET
END_PROPERTY

METHOD Mr_Read : BOOL
VAR_INPUT
END_VAR
IF nState = STATE_WAIT_CMD THEN
	nState := STATE_READ1;
END_IF
END_METHOD

END_PROGRAM

// ---- POUs/Program/IP233.TcPOU
PROGRAM IP233
VAR
	timer				: TON;
	nState				: INT := STATE_INIT;
	
	fbInit233_01_5350			: FB_InitPM;
	fbInit233_03_5350			: FB_InitPM;
	fbInit233_05_5350			: FB_InitPM;
	fbInit233_07_5350			: FB_InitPM;
	fbInit233_08_5350			: FB_InitPM;
	
	fbRead233_01_5350			: FB_ReadPM5350;
	fbRead233_03_5350			: FB_ReadPM5350;
	fbRead233_05_5350			: FB_ReadPM5350;
	fbRead233_07_5350			: FB_ReadPM5350;
	fbRead233_08_5350			: FB_ReadPM5350;
	
	fbInit233_02_5500			: FB_InitPM;
	fbInit233_04_5500			: FB_InitPM;
	fbInit233_06_5500			: FB_InitPM;
	
	fbRead233_02_5500			: FB_ReadPM5500;
	fbRead233_04_5500			: FB_ReadPM5500;
	fbRead233_06_5500			: FB_ReadPM5500;
	
	nCount						: DINT;
END_VAR

VAR CONSTANT
	STATE_INIT			:	INT		:= 0;
	STATE_WAIT_CMD		: 	INT		:= 5;
	STATE_READ1			:	INT		:= 10;
	STATE_READ3			:	INT		:= 30;
	STATE_READ5			:	INT		:= 50;
	STATE_READ7			:	INT		:= 70;
	STATE_READ8			:	INT		:= 80;
	STATE_READ2			:	INT		:= 20;
	STATE_READ4			:	INT		:= 40;
	STATE_READ6			:	INT		:= 60;
END_VAR

CASE nState OF
	STATE_INIT:
		fbInit233_01_5350(	sIpAddress	:= '10.91.37.233',
							nPort		:= 502,
							nUnitID		:= 1,
							PM			:= pmDev.DB03_01_5350);
		fbInit233_03_5350(	sIpAddress	:= '10.91.37.233',
							nPort		:= 502,
							nUnitID		:= 3,
							PM			:= pmDev.DB03_03_5350);
		fbInit233_05_5350(	sIpAddress	:= '10.91.37.233',
							nPort		:= 502,
							nUnitID		:= 5,
							PM			:= pmDev.DB03_05_5350);
		fbInit233_07_5350(	sIpAddress	:= '10.91.37.233',
							nPort		:= 502,
							nUnitID		:= 7,
							PM			:= pmDev.DB03_07_5350);
		fbInit233_08_5350(	sIpAddress	:= '10.91.37.233',
							nPort		:= 502,
							nUnitID		:= 8,
							PM			:= pmDev.DB03_08_5350);
							
		fbInit233_02_5500(	sIpAddress	:= '10.91.37.233',
							nPort		:= 502,
							nUnitID		:= 2,
							PM			:= pmDev.DB03_02_5500);
		fbInit233_04_5500(	sIpAddress	:= '10.91.37.233',
							nPort		:= 502,
							nUnitID		:= 4,
							PM			:= pmDev.DB03_04_5500);
		fbInit233_06_5500(	sIpAddress	:= '10.91.37.233',
							nPort		:= 502,
							nUnitID		:= 6,
							PM			:= pmDev.DB03_06_5500);
								
		timer(In:=TRUE, PT:= TIME_INIT);
		IF timer.Q THEN
			timer(In:= FALSE);
			nState	:= STATE_WAIT_CMD;
		END_IF
		
	STATE_WAIT_CMD:
			;
			
	STATE_READ1:
		fbRead233_01_5350(
			bExecute:=TRUE,
			PM:= pmDev.DB03_01_5350);
		IF NOT fbRead233_01_5350.Q THEN
			nState	:= STATE_READ3;
			fbRead233_01_5350(
				bExecute:=FALSE,
				PM:= pmDev.DB03_01_5350);
		END_IF
		
	STATE_READ3:
		fbRead233_03_5350(
			bExecute:=TRUE,
			PM:= pmDev.DB03_03_5350);
		IF NOT fbRead233_03_5350.Q THEN
			nState	:= STATE_READ5;
			fbRead233_03_5350(
				bExecute:=FALSE,
				PM:= pmDev.DB03_03_5350);
		END_IF	
	
	STATE_READ5:
		fbRead233_05_5350(
			bExecute:=TRUE,
			PM:= pmDev.DB03_05_5350);
		IF NOT fbRead233_05_5350.Q THEN
			nState	:= STATE_READ7;
			fbRead233_05_5350(
				bExecute:=FALSE,
				PM:= pmDev.DB03_05_5350);
		END_IF	
		
	STATE_READ7:
		fbRead233_07_5350(
			bExecute:=TRUE,
			PM:= pmDev.DB03_07_5350);
		IF NOT fbRead233_07_5350.Q THEN
			nState	:= STATE_READ8;
			fbRead233_07_5350(
				bExecute:=FALSE,
				PM:= pmDev.DB03_07_5350);
		END_IF	
		
	STATE_READ8:
		fbRead233_08_5350(
			bExecute:=TRUE,
			PM:= pmDev.DB03_08_5350);
		IF NOT fbRead233_08_5350.Q THEN
			nState	:= STATE_READ2;
			fbRead233_08_5350(
				bExecute:=FALSE,
				PM:= pmDev.DB03_08_5350);
		END_IF	
		
	STATE_READ2:
		fbRead233_02_5500(
			bExecute:=TRUE,
			PM:= pmDev.DB03_02_5500);
		IF NOT fbRead233_02_5500.Q THEN
			nState	:= STATE_READ4;
			fbRead233_02_5500(
				bExecute:=FALSE,
				PM:= pmDev.DB03_02_5500);
		END_IF
	STATE_READ4:
		fbRead233_04_5500(
			bExecute:=TRUE,
			PM:= pmDev.DB03_04_5500);
		IF NOT fbRead233_04_5500.Q THEN
			nState	:= STATE_READ6;
			fbRead233_04_5500(
				bExecute:=FALSE,
				PM:= pmDev.DB03_04_5500);
		END_IF
	
	STATE_READ6:
		fbRead233_06_5500(
			bExecute:=TRUE,
			PM:= pmDev.DB03_06_5500);
		IF NOT fbRead233_06_5500.Q THEN
			nState	:= STATE_WAIT_CMD;
			fbRead233_06_5500(
				bExecute:=FALSE,
				PM:= pmDev.DB03_06_5500);
		END_IF
		
END_CASE

PROPERTY Busy : Bool
GET
Busy := nState <> STATE_WAIT_CMD;
END_GET
END_PROPERTY

METHOD Mr_Read : BOOL
VAR_INPUT
END_VAR
IF nState = STATE_WAIT_CMD THEN
	nState := STATE_READ1;
END_IF
END_METHOD

END_PROGRAM

// ---- POUs/Program/IP234.TcPOU
PROGRAM IP234
VAR
	timer				: TON;
	nState				: INT := STATE_INIT;
	fbInit234_01_5350			: FB_InitPM;
	fbInit234_03_5350			: FB_InitPM;
	fbInit234_05_5350			: FB_InitPM;
	fbInit234_07_5350			: FB_InitPM;
	fbInit234_08_5350			: FB_InitPM;
	
	fbRead234_01_5350			: FB_ReadPM5350;
	fbRead234_03_5350			: FB_ReadPM5350;
	fbRead234_05_5350			: FB_ReadPM5350;
	fbRead234_07_5350			: FB_ReadPM5350;
	fbRead234_08_5350			: FB_ReadPM5350;

	fbInit234_02_5500			: FB_InitPM;
	fbInit234_04_5500			: FB_InitPM;
	fbInit234_06_5500			: FB_InitPM;

	fbRead234_02_5500			: FB_ReadPM5500;
	fbRead234_04_5500			: FB_ReadPM5500;
	fbRead234_06_5500			: FB_ReadPM5500;
	
	nCount						: DINT;
END_VAR

VAR CONSTANT
	STATE_INIT			:	INT		:= 0;
	STATE_WAIT_CMD		: 	INT		:= 5;
	STATE_READ1			:	INT		:= 10;
	STATE_READ3			:	INT		:= 30;
	STATE_READ5			:	INT		:= 50;
	STATE_READ7			:	INT		:= 70;
	STATE_READ8			:	INT		:= 80;
	STATE_READ2			:	INT		:= 20;
	STATE_READ4			:	INT		:= 40;
	STATE_READ6			:	INT		:= 60;
END_VAR

CASE nState OF
	STATE_INIT:
		fbInit234_01_5350(	sIpAddress	:= '10.91.37.234',
							nPort		:= 502,
							nUnitID		:= 1,
							PM			:= pmDev.DB04_01_5350);
		fbInit234_03_5350(	sIpAddress	:= '10.91.37.234',
							nPort		:= 502,
							nUnitID		:= 3,
							PM			:= pmDev.DB04_03_5350);
		fbInit234_05_5350(	sIpAddress	:= '10.91.37.234',
							nPort		:= 502,
							nUnitID		:= 5,
							PM			:= pmDev.DB04_05_5350);
		fbInit234_07_5350(	sIpAddress	:= '10.91.37.234',
							nPort		:= 502,
							nUnitID		:= 7,
							PM			:= pmDev.DB04_07_5350);
		fbInit234_08_5350(	sIpAddress	:= '10.91.37.234',
							nPort		:= 502,
							nUnitID		:= 8,
							PM			:= pmDev.DB04_08_5350);
							
		fbInit234_02_5500(	sIpAddress	:= '10.91.37.234',
							nPort		:= 502,
							nUnitID		:= 2,
							PM			:= pmDev.DB04_02_5500);
		fbInit234_04_5500(	sIpAddress	:= '10.91.37.234',
							nPort		:= 502,
							nUnitID		:= 4,
							PM			:= pmDev.DB04_04_5500);
		fbInit234_06_5500(	sIpAddress	:= '10.91.37.234',
							nPort		:= 502,
							nUnitID		:= 6,
							PM			:= pmDev.DB04_06_5500);
								
		timer(In:=TRUE, PT:= TIME_INIT);
		IF timer.Q THEN
			timer(In:=FALSE);
			nState	:= STATE_WAIT_CMD;
		END_IF
		
	STATE_WAIT_CMD:
			;
			
	STATE_READ1:
		fbRead234_01_5350(
			bExecute:=TRUE,
			PM:= pmDev.DB04_01_5350);
		IF NOT fbRead234_01_5350.Q THEN
			nState	:= STATE_READ3;
			fbRead234_01_5350(
				bExecute:=FALSE,
				PM:= pmDev.DB04_01_5350);
		END_IF
		
	STATE_READ3:
		fbRead234_03_5350(
			bExecute:=TRUE,
			PM:= pmDev.DB04_03_5350);
		IF NOT fbRead234_03_5350.Q THEN
			nState	:= STATE_READ5;
			fbRead234_03_5350(
				bExecute:=FALSE,
				PM:= pmDev.DB04_03_5350);
		END_IF	
	
	STATE_READ5:
		fbRead234_05_5350(
			bExecute:=TRUE,
			PM:= pmDev.DB04_05_5350);
		IF NOT fbRead234_05_5350.Q THEN
			nState	:= STATE_READ7;
			fbRead234_05_5350(
				bExecute:=FALSE,
				PM:= pmDev.DB04_05_5350);
		END_IF	
		
	STATE_READ7:
		fbRead234_07_5350(
			bExecute:=TRUE,
			PM:= pmDev.DB04_07_5350);
		IF NOT fbRead234_07_5350.Q THEN
			nState	:= STATE_READ8;
			fbRead234_07_5350(
				bExecute:=FALSE,
				PM:= pmDev.DB04_07_5350);
		END_IF	
		
	STATE_READ8:
		fbRead234_08_5350(
			bExecute:=TRUE,
			PM:= pmDev.DB04_08_5350);
		IF NOT fbRead234_08_5350.Q THEN
			nState	:= STATE_READ2;
			fbRead234_08_5350(
				bExecute:=FALSE,
				PM:= pmDev.DB04_08_5350);
		END_IF	
		
	STATE_READ2:
		fbRead234_02_5500(
			bExecute:=TRUE,
			PM:= pmDev.DB04_02_5500);
		IF NOT fbRead234_02_5500.Q THEN
			nState	:= STATE_READ4;
			fbRead234_02_5500(
				bExecute:=FALSE,
				PM:= pmDev.DB04_02_5500);
		END_IF
	STATE_READ4:
		fbRead234_04_5500(
			bExecute:=TRUE,
			PM:= pmDev.DB04_04_5500);
		IF NOT fbRead234_04_5500.Q THEN
			nState	:= STATE_READ6;
			fbRead234_04_5500(
				bExecute:=FALSE,
				PM:= pmDev.DB04_04_5500);
		END_IF
	
	STATE_READ6:
		fbRead234_06_5500(
			bExecute:=TRUE,
			PM:= pmDev.DB04_06_5500);
		IF NOT fbRead234_06_5500.Q THEN
			nState	:= STATE_WAIT_CMD;
			fbRead234_06_5500(
				bExecute:=FALSE,
				PM:= pmDev.DB04_06_5500);
		END_IF
	
END_CASE

PROPERTY Busy : Bool
GET
Busy := nState <> STATE_WAIT_CMD;
END_GET
END_PROPERTY

METHOD Mr_Read : BOOL
VAR_INPUT
END_VAR
IF nState = STATE_WAIT_CMD THEN
	nState := STATE_READ1;
END_IF
END_METHOD

END_PROGRAM

// ---- POUs/Program/Ip235.TcPOU
PROGRAM IP235
VAR
	timer				: TON;
	nState				: INT := STATE_INIT;
	
	fbInit235_01_5350			: FB_InitPM;
	fbInit235_02_5350			: FB_InitPM;
	fbInit235_03_5350			: FB_InitPM;
	fbInit235_05_5350			: FB_InitPM;
	fbInit235_07_5350			: FB_InitPM;
	fbInit235_09_5350			: FB_InitPM;
	fbInit235_21_5350			: FB_InitPM;
	fbInit235_22_5350			: FB_InitPM;
	
	fbRead235_01_5350			: FB_ReadPM5350;
	fbRead235_02_5350			: FB_ReadPM5350;
	fbRead235_03_5350			: FB_ReadPM5350;
	fbRead235_05_5350			: FB_ReadPM5350;
	fbRead235_07_5350			: FB_ReadPM5350;
	fbRead235_09_5350			: FB_ReadPM5350;
	fbRead235_21_5350			: FB_ReadPM5350;
	fbRead235_22_5350			: FB_ReadPM5350;
	
	fbInit235_04_5500			: FB_InitPM;
	fbInit235_06_5500			: FB_InitPM;
	fbInit235_08_5500			: FB_InitPM;
	fbInit235_10_5500			: FB_InitPM;
	
	fbRead235_04_5500			: FB_ReadPM5500;
	fbRead235_06_5500			: FB_ReadPM5500;
	fbRead235_08_5500			: FB_ReadPM5500;
	fbRead235_10_5500			: FB_ReadPM5500;
	
	nCount						: DINT;
END_VAR

VAR CONSTANT
	STATE_INIT			:	INT		:= 0;
	STATE_WAIT_CMD		: 	INT		:= 5;
	STATE_READ1			:	INT		:= 10;
	STATE_READ2			:	INT		:= 20;
	STATE_READ3			:	INT		:= 30;
	STATE_READ5			:	INT		:= 50;
	STATE_READ7			:	INT		:= 70;
	STATE_READ9			:	INT		:= 90;
	STATE_READ21		:	INT		:= 210;
	STATE_READ22		:	INT		:= 220;
	STATE_READ4			:	INT		:= 40;
	STATE_READ6			:	INT		:= 60;
	STATE_READ8			:	INT		:= 80;
	STATE_READ10		:	INT		:= 100;
END_VAR

CASE nState OF
	STATE_INIT:
		fbInit235_01_5350(	sIpAddress	:= '10.91.37.235',
							nPort		:= 502,
							nUnitID		:= 1,
							PM			:= pmDev.DB05_01_5350);
		fbInit235_02_5350(	sIpAddress	:= '10.91.37.235',
							nPort		:= 502,
							nUnitID		:= 2,
							PM			:= pmDev.DB05_02_5350);
		fbInit235_03_5350(	sIpAddress	:= '10.91.37.235',
							nPort		:= 502,
							nUnitID		:= 3,
							PM			:= pmDev.DB05_03_5350);
		fbInit235_05_5350(	sIpAddress	:= '10.91.37.235',
							nPort		:= 502,
							nUnitID		:= 5,
							PM			:= pmDev.DB05_05_5350);
		fbInit235_07_5350(	sIpAddress	:= '10.91.37.235',
							nPort		:= 502,
							nUnitID		:= 7,
							PM			:= pmDev.DB05_07_5350);
		fbInit235_09_5350(	sIpAddress	:= '10.91.37.235',
							nPort		:= 502,
							nUnitID		:= 9,
							PM			:= pmDev.DB05_09_5350);
							
		fbInit235_21_5350(	sIpAddress	:= '10.91.37.235',
							nPort		:= 502,
							nUnitID		:= 21,
							PM			:= pmDev.DB05_21_5350);
							
		fbInit235_22_5350(	sIpAddress	:= '10.91.37.235',
							nPort		:= 502,
							nUnitID		:= 22,
							PM			:= pmDev.DB05_22_5350);	
							
		fbInit235_04_5500(	sIpAddress	:= '10.91.37.235',
							nPort		:= 502,
							nUnitID		:= 4,
							PM			:= pmDev.DB05_04_5500);
		fbInit235_06_5500(	sIpAddress	:= '10.91.37.235',
							nPort		:= 502,
							nUnitID		:= 6,
							PM			:= pmDev.DB05_06_5500);
		fbInit235_08_5500(	sIpAddress	:= '10.91.37.235',
							nPort		:= 502,
							nUnitID		:= 8,
							PM			:= pmDev.DB05_08_5500);
		fbInit235_10_5500(	sIpAddress	:= '10.91.37.235',
							nPort		:= 502,
							nUnitID		:= 10,
							PM			:= pmDev.DB05_10_5500);
							
		timer(In:=TRUE, PT:= TIME_INIT);
		IF timer.Q THEN
			timer(In:=FALSE);
			nState	:= STATE_WAIT_CMD;
		END_IF
		
	STATE_WAIT_CMD:
		;
		
	STATE_READ1:
		fbRead235_01_5350(
			bExecute:=TRUE,
			PM:= pmDev.DB05_01_5350);
		IF NOT fbRead235_01_5350.Q THEN
			nState	:= STATE_READ2;
			fbRead235_01_5350(
				bExecute:=FALSE,
				PM:= pmDev.DB05_01_5350);
		END_IF
		
	STATE_READ2:
		fbRead235_02_5350(
			bExecute:=TRUE,
			PM:= pmDev.DB05_02_5350);
		IF NOT fbRead235_02_5350.Q THEN
			nState	:= STATE_READ3;
			fbRead235_02_5350(
				bExecute:=FALSE,
				PM:= pmDev.DB05_02_5350);
		END_IF	
	
	STATE_READ3:
		fbRead235_03_5350(
			bExecute:=TRUE,
			PM:= pmDev.DB05_03_5350);
		IF NOT fbRead235_03_5350.Q THEN
			nState	:= STATE_READ5;
			fbRead235_03_5350(
				bExecute:=FALSE,
				PM:= pmDev.DB05_03_5350);
		END_IF	
		
	STATE_READ5:
		fbRead235_05_5350(
			bExecute:=TRUE,
			PM:= pmDev.DB05_05_5350);
		IF NOT fbRead235_05_5350.Q THEN
			nState	:= STATE_READ7;
			fbRead235_05_5350(
				bExecute:=FALSE,
				PM:= pmDev.DB05_05_5350);
		END_IF	
		
	STATE_READ7:
		fbRead235_07_5350(
			bExecute:=TRUE,
			PM:= pmDev.DB05_07_5350);
		IF NOT fbRead235_07_5350.Q THEN
			nState	:= STATE_READ9;
			fbRead235_07_5350(
				bExecute:=FALSE,
				PM:= pmDev.DB05_07_5350);
		END_IF	
		
	STATE_READ9:
		fbRead235_09_5350(
			bExecute:=TRUE,
			PM:= pmDev.DB05_09_5350);
		IF NOT fbRead235_09_5350.Q THEN
			nState	:= STATE_READ21;
			fbRead235_09_5350(
				bExecute:=FALSE,
				PM:= pmDev.DB05_09_5350);
		END_IF	
		
	STATE_READ21:
		fbRead235_21_5350(
			bExecute:=TRUE,
			PM:= pmDev.DB05_21_5350);
		IF NOT fbRead235_21_5350.Q THEN
			nState	:= STATE_READ22;
			fbRead235_21_5350(
				bExecute:=FALSE,
				PM:= pmDev.DB05_21_5350);
		END_IF	
		
	STATE_READ22:
		fbRead235_22_5350(
			bExecute:=TRUE,
			PM:= pmDev.DB05_22_5350);
		IF NOT fbRead235_22_5350.Q THEN
			nState	:= STATE_READ4;
			fbRead235_22_5350(
				bExecute:=FALSE,
				PM:= pmDev.DB05_22_5350);
		END_IF	
		
	STATE_READ4:
		fbRead235_04_5500(
			bExecute:=TRUE,
			PM:= pmDev.DB05_04_5500);
		IF NOT fbRead235_04_5500.Q THEN
			nState	:= STATE_READ6;
			fbRead235_04_5500(
				bExecute:=FALSE,
				PM:= pmDev.DB05_04_5500);
		END_IF
	STATE_READ6:
		fbRead235_06_5500(
			bExecute:=TRUE,
			PM:= pmDev.DB05_06_5500);
		IF NOT fbRead235_06_5500.Q THEN
			nState	:= STATE_READ8;
			fbRead235_06_5500(
				bExecute:=FALSE,
				PM:= pmDev.DB05_06_5500);
		END_IF
	
	STATE_READ8:
		fbRead235_08_5500(
			bExecute:=TRUE,
			PM:= pmDev.DB05_08_5500);
		IF NOT fbRead235_08_5500.Q THEN
			nState	:= STATE_READ10;
			fbRead235_08_5500(
				bExecute:=FALSE,
				PM:= pmDev.DB05_08_5500);
		END_IF
	STATE_READ10:
		fbRead235_10_5500(
			bExecute:=TRUE,
			PM:= pmDev.DB05_10_5500);
		IF NOT fbRead235_10_5500.Q THEN
			nState	:= STATE_WAIT_CMD;
			fbRead235_10_5500(
				bExecute:=FALSE,
				PM:= pmDev.DB05_10_5500);
		END_IF
		
END_CASE

PROPERTY Busy : Bool
GET
Busy := nState <> STATE_WAIT_CMD;
END_GET
END_PROPERTY

METHOD Mr_Read : BOOL
VAR_INPUT
END_VAR
IF nState = STATE_WAIT_CMD THEN
	nState := STATE_READ1;
END_IF
END_METHOD

END_PROGRAM

// ---- POUs/Program/IP236.TcPOU
PROGRAM IP236
VAR
	timer				: TON;
	nState				: INT := STATE_INIT;
	
	fbInit236_01_5500			: FB_InitPM;
	fbInit236_02_5500			: FB_InitPM;
	fbInit236_03_5500			: FB_InitPM;
	fbInit236_04_5500			: FB_InitPM;
	fbInit236_05_5500			: FB_InitPM;
	fbInit236_06_5500			: FB_InitPM;
	fbInit236_07_5500			: FB_InitPM;
	fbInit236_08_5500			: FB_InitPM;
	fbInit236_11_5500			: FB_InitPM;
	fbInit236_33_5500			: FB_InitPM;
	fbInit236_38_5500			: FB_InitPM;
	
	fbRead236_01_5500			: FB_ReadPM5500;
	fbRead236_02_5500			: FB_PM_ION_9000;
	
	//Update 29-08-2022
	fbRead236_03_5500			: FB_ReadPM5350;
	
	fbRead236_04_5500			: FB_PM_ION_9000;
	
	//Update 29-08-2022
	fbRead236_05_5500			: FB_ReadPM5350;
	//Update 29-08-2022
	fbRead236_06_5500			: FB_ReadPM5350;
	
	
	fbRead236_07_5500			: FB_ReadPM5500;
	fbRead236_08_5500			: FB_ReadPM5500;
	fbRead236_11_5500			: FB_ReadPM5500;
	fbRead236_33_5500			: FB_ReadPM5500;
	fbRead236_38_5500			: FB_ReadPM5500;
	
	nCount						: DINT;
END_VAR

VAR CONSTANT
	STATE_INIT			:	INT		:= 0;
	STATE_WAIT_CMD		: 	INT		:= 5;
	STATE_READ1			:	INT		:= 10;
	STATE_READ2			:	INT		:= 20;
	STATE_READ3			:	INT		:= 30;
	STATE_READ4			:	INT		:= 40;
	STATE_READ5			:	INT		:= 50;
	STATE_READ6			:	INT		:= 60;
	STATE_READ7			:	INT		:= 70;
	STATE_READ8			:	INT		:= 80;
	STATE_READ11		:	INT		:= 110;
	STATE_READ33		:	INT		:= 330;
	STATE_READ38		:	INT		:= 380;
END_VAR

CASE nState OF
	STATE_INIT:
		fbInit236_01_5500(	sIpAddress	:= '10.91.37.236',
							nPort		:= 502,
							nUnitID		:= 1,
							PM			:= pmDev.DB06_01_5500);
		fbInit236_02_5500(	sIpAddress	:= '10.91.37.230',
							nPort		:= 502,
							nUnitID		:= 255,
							PM			:= pmDev.DB06_02_5500);
		fbInit236_03_5500(	sIpAddress	:= '10.91.37.236',
							nPort		:= 502,
							nUnitID		:= 3,
							PM			:= pmDev.DB06_03_5500);
		fbInit236_04_5500(	sIpAddress	:= '10.91.37.229',
							nPort		:= 502,
							nUnitID		:= 255,
							PM			:= pmDev.DB06_04_5500);
		fbInit236_05_5500(	sIpAddress	:= '10.91.37.236',
							nPort		:= 502,
							nUnitID		:= 5,
							PM			:= pmDev.DB06_05_5500);
							
		fbInit236_06_5500(	sIpAddress	:= '10.91.37.236',
							nPort		:= 502,
							nUnitID		:= 6,
							PM			:= pmDev.DB06_06_5500);
							
		fbInit236_07_5500(	sIpAddress	:= '10.91.37.236',
							nPort		:= 502,
							nUnitID		:= 7,
							PM			:= pmDev.DB06_07_5500);
							
		fbInit236_08_5500(	sIpAddress	:= '10.91.37.236',
							nPort		:= 502,
							nUnitID		:= 8,
							PM			:= pmDev.DB06_08_5500);
							
		fbInit236_11_5500(	sIpAddress	:= '10.91.37.236',
							nPort		:= 502,
							nUnitID		:= 11,
							PM			:= pmDev.DB06_11_5500);
							
		fbInit236_33_5500(	sIpAddress	:= '10.91.37.236',
							nPort		:= 502,
							nUnitID		:= 33,
							PM			:= pmDev.DB06_33_5500);
							
		fbInit236_38_5500(	sIpAddress	:= '10.91.37.236',
							nPort		:= 502,
							nUnitID		:= 38,
							PM			:= pmDev.DB06_38_5500);
		
		timer(In:=TRUE, PT:= TIME_INIT);
		IF timer.Q THEN
			timer(In := FALSE);
			nState	:= STATE_WAIT_CMD;
		END_IF
		
	STATE_WAIT_CMD:
		;
		
	STATE_READ1:
		fbRead236_01_5500(
			bExecute:=TRUE,
			PM:= pmDev.DB06_01_5500);
		IF NOT fbRead236_01_5500.Q THEN
			nState	:= STATE_READ2;
			fbRead236_01_5500(
				bExecute:=FALSE,
				PM:= pmDev.DB06_01_5500);
		END_IF
		
	STATE_READ2:
		fbRead236_02_5500(
			bExecute:=TRUE,
			PM:= pmDev.DB06_02_5500);
		IF NOT fbRead236_02_5500.Q THEN
			nState	:= STATE_READ3;
			fbRead236_02_5500(
				bExecute:=FALSE,
				PM:= pmDev.DB06_02_5500);
		END_IF	
	
	STATE_READ3:
	
		fbRead236_03_5500(
			bExecute:=TRUE,
			PM:= pmDev.DB06_03_5500);
		IF NOT fbRead236_03_5500.Q THEN
			nState	:= STATE_READ4;
			fbRead236_03_5500(
				bExecute:=FALSE,
				PM:= pmDev.DB06_03_5500);
		END_IF	
		
	STATE_READ4:
		fbRead236_04_5500(
			bExecute:=TRUE,
			PM:= pmDev.DB06_04_5500);
		IF NOT fbRead236_04_5500.Q THEN
			nState	:= STATE_READ5;
			fbRead236_04_5500(
				bExecute:=FALSE,
				PM:= pmDev.DB06_04_5500);
		END_IF	
		
	STATE_READ5:
	
		fbRead236_05_5500(
			bExecute:=TRUE,
			PM:= pmDev.DB06_05_5500);
		IF NOT fbRead236_05_5500.Q THEN
			nState	:= STATE_READ6;
			fbRead236_05_5500(
				bExecute:=FALSE,
				PM:= pmDev.DB06_06_5500);
		END_IF	
		
	STATE_READ6:
	
		
		fbRead236_06_5500(
			bExecute:=TRUE,
			PM:= pmDev.DB06_06_5500);
		IF NOT fbRead236_06_5500.Q THEN
			nState	:= STATE_READ7;
			fbRead236_06_5500(
				bExecute:=FALSE,
				PM:= pmDev.DB06_06_5500);
		END_IF	
		
	STATE_READ7:
		fbRead236_07_5500(
			bExecute:=TRUE,
			PM:= pmDev.DB06_07_5500);
		IF NOT fbRead236_07_5500.Q THEN
			nState	:= STATE_READ8;
			fbRead236_07_5500(
				bExecute:=FALSE,
				PM:= pmDev.DB06_07_5500);
		END_IF
		
	STATE_READ8:
		fbRead236_08_5500(
			bExecute:=TRUE,
			PM:= pmDev.DB06_08_5500);
		IF NOT fbRead236_08_5500.Q THEN
			nState	:= STATE_READ11;
			fbRead236_08_5500(
				bExecute:=FALSE,
				PM:= pmDev.DB06_08_5500);
		END_IF
		
	STATE_READ11:
		fbRead236_11_5500(
			bExecute:=TRUE,
			PM:= pmDev.DB06_11_5500);
		IF NOT fbRead236_11_5500.Q THEN
			nState	:= STATE_READ33;
			fbRead236_11_5500(
				bExecute:=FALSE,
				PM:= pmDev.DB06_11_5500);
		END_IF
		
	STATE_READ33:
		fbRead236_33_5500(
			bExecute:=TRUE,
			PM:= pmDev.DB06_33_5500);
		IF NOT fbRead236_33_5500.Q THEN
			nState	:= STATE_READ38;
			fbRead236_33_5500(
				bExecute:=FALSE,
				PM:= pmDev.DB06_33_5500);
		END_IF
		
	STATE_READ38:
		fbRead236_38_5500(
			bExecute:=TRUE,
			PM:= pmDev.DB06_38_5500);
		IF NOT fbRead236_38_5500.Q THEN
			nState	:= STATE_WAIT_CMD;
			fbRead236_38_5500(
				bExecute:=FALSE,
				PM:= pmDev.DB06_38_5500);
		END_IF
		
END_CASE

PROPERTY Busy : Bool
GET
Busy := nState <> STATE_WAIT_CMD;
END_GET
END_PROPERTY

METHOD Mr_Read : BOOL
VAR_INPUT
END_VAR
IF nState = STATE_WAIT_CMD THEN
	nState := STATE_READ1;
END_IF
END_METHOD

END_PROGRAM

// ---- POUs/Metters/FB_PM_ION_9000.TcPOU
FUNCTION_BLOCK FB_PM_ION_9000

VAR_INPUT
	bExecute	: BOOL;
END_VAR

VAR_OUTPUT
	Q			: BOOL;
END_VAR

VAR_IN_OUT
	PM		:	ST_PowerMeter;
END_VAR

VAR
	fbReadRegs      	: FB_MBReadRegs;
	nState				: INT;
	nQuantity       	: WORD:=125;
	nMBAddr             : WORD:=1;
	bDoReading			: BOOL;
	
	bReadRegsBusy   	: BOOL;
	bReadRegsError  	: BOOL;
	nReadRegsErrorId    : UDINT;
	nReadRegsCount  	: UDINT;
	
	nCount				: DINT;
	rTrigExecute		: R_TRIG;
	

	nMBAddressDestAddr	: WORD;
	arrRawData			: ARRAY[0..124] OF WORD;
	iloop				: INT;
	offset				: UDINT;
END_VAR

VAR CONSTANT
	STATE_IDLE			:	INT		:=0;
	STATE_INIT			:	INT		:=5;
	STATE_PREPARE		:	INT		:=10;
	STATE_READ			:	INT		:=20;
	STATE_ERROR			:	INT		:=30;
	STATE_CALCULATE		:	INT		:= 90;
END_VAR
VAR PERSISTENT
	validEnvergyIntoLoad : LREAL;
END_VAR

rTrigExecute(clk:= bExecute);
IF rTrigExecute.Q THEN
	nState		:= STATE_INIT;
END_IF

CASE nState OF
STATE_IDLE:
	nCount	:=	nCount + 1;
	
STATE_INIT:
	nMBAddr			:= 0;
	Q				:= TRUE;
	bDoReading		:= TRUE;
	nState			:= STATE_PREPARE;
	nQuantity		:= 125;
	
STATE_PREPARE:
	IF nMBAddr=0 THEN
		nMBAddr	:= 1;
	ELSIF nMBAddr > 3300 AND nMBAddr < 20000   THEN
		nMBAddr	:= 21296;
	ELSE
		nMBAddr	:= nMBAddr + 125;
	END_IF
	
	
	IF  nMBAddr > 21500 THEN
		nState		:= STATE_CALCULATE;
	ELSE 
		nState				:= STATE_READ;
		fbReadRegs.bExecute	:= FALSE;
	END_IF
STATE_READ:
	IF nMBAddr <20000 THEN
		nMBAddressDestAddr := nMBAddr;
	ELSIF nMBAddr >= 21296 THEN
		nMBAddressDestAddr := nMBAddr - 15000 ;		
	END_IF
	fbReadRegs (
			sIPAddr		:= PM.Conn.sIPAddress,
			nTCPPort	:= PM.Conn.nPort,
			nUnitID		:= PM.Conn.nUnitID,
			nQuantity	:= nQuantity,
			nMBAddr		:= nMBAddr,
			cbLength	:= nQuantity*2,
			pDestAddr	:= ADR(PM.RawData) + nMBAddressDestAddr*2 + 2,
			bExecute	:= TRUE,
			bBusy		=> bReadRegsBusy,
			bError		=> bReadRegsError,
			nErrId		=> nReadRegsErrorId,
			cbRead		=> nReadRegsCount
		);
	IF NOT fbReadRegs.bBusy THEN
		fbReadRegs(bExecute:= FALSE);
		nState			:= STATE_PREPARE;
	END_IF
STATE_CALCULATE:
	//PM.Basic.Current_Unbalane_A 		:= F_Read_RegFloat32(PM:= PM, address:= ION9000_E_Current_Unbalane_A);
	//PM.Basic.Current_Unbalane_B 		:= F_Read_RegFloat32(PM:= PM, address:=E_PM5350.E_Current_Unbalane_B);
	//PM.Basic.Current_Unbalane_C 		:= F_Read_RegFloat32(PM:= PM, address:=E_PM5350.E_Current_Unbalane_C);
	PM.Basic.Current_Unbalane_Worst 	:= F_Read_RegFloat32(PM:= PM, address:= ION9000_E_Current_Unbalane_Worst);
	//PM.Basic.Current_Unbalane_AB 		:= F_Read_RegFloat32(PM:= PM, address:=E_PM5350.E_Current_Unbalane_AB);
	//	PM.Basic.Current_Unbalane_BC		:= F_Read_RegFloat32(PM:= PM, address:=E_PM5350.E_Current_Unbalane_BC);
	//	PM.Basic.Current_Unbalane_CA 		:= F_Read_RegFloat32(PM:= PM, address:=E_PM5350.E_Current_Unbalane_CA);
	//	PM.Basic.Current_Unbalane_LL_Worst 	:= F_Read_RegFloat32(PM:= PM, address:=E_PM5350.E_Current_Unbalane_LL_Worst);
	//	PM.Basic.Current_Unbalane_AN 		:= F_Read_RegFloat32(PM:= PM, address:=E_PM5350.E_Current_Unbalane_AN);
	//	PM.Basic.Current_Unbalane_BN 		:= F_Read_RegFloat32(PM:= PM, address:=E_PM5350.E_Current_Unbalane_BN);
	//	PM.Basic.Current_Unbalane_CN 		:= F_Read_RegFloat32(PM:= PM, address:=E_PM5350.E_Current_Unbalane_CN);
	//PM.Basic.Current_Unbalane_LN_Worst	:= F_Read_RegFloat32(PM:= PM, address:=ION9000_E_Current_Unbalane_LN_Worst);
	PM.Basic.Real_PowerA 				:= F_Read_RegFloat32(PM:= PM, address:=ION9000_E_Real_PowerA)/1000;//kw
	PM.Basic.Real_PowerB 				:= F_Read_RegFloat32(PM:= PM, address:=ION9000_E_Real_PowerB)/1000;
	PM.Basic.Real_PowerC 				:= F_Read_RegFloat32(PM:= PM, address:=ION9000_E_Real_PowerC)/1000;
	PM.Basic.Real_PowerTotal 			:= F_Read_RegFloat32(PM:= PM, address:=ION9000_E_Real_PowerTotal)/1000;
	
	PM.Basic.Reactive_PowerA 			:= F_Read_RegFloat32(PM:= PM, address:=ION9000_E_Reactive_PowerA)/1000;
	PM.Basic.Reactive_PowerB 			:= F_Read_RegFloat32(PM:= PM, address:=ION9000_E_Reactive_PowerB)/1000;
	PM.Basic.Reactive_PowerC 			:= F_Read_RegFloat32(PM:= PM, address:=ION9000_E_Reactive_PowerC)/1000;
	PM.Basic.Reactive_PowerTotal 		:= F_Read_RegFloat32(PM:= PM, address:=ION9000_E_Reactive_PowerTotal)/1000;
	
	PM.Basic.Apparent_PowerA 			:= F_Read_RegFloat32(PM:= PM, address:=ION9000_E_Apparent_PowerA)/1000;
	PM.Basic.Apparent_PowerB 			:= F_Read_RegFloat32(PM:= PM, address:=ION9000_E_Apparent_PowerB)/1000;
	PM.Basic.Apparent_PowerC 			:= F_Read_RegFloat32(PM:= PM, address:=ION9000_E_Apparent_PowerC)/1000;
	PM.Basic.Apparent_PowerTotal 		:= F_Read_RegFloat32(PM:= PM, address:=ION9000_E_Apparent_PowerTotal)/1000;
	
	PM.Basic.Voltage_AB 			:= F_Read_RegFloat32(PM:= PM, address:=ION9000_E_Voltage_AB);
	PM.Basic.Voltage_BC 			:= F_Read_RegFloat32(PM:= PM, address:=ION9000_E_Voltage_BC);
	PM.Basic.Voltage_CA 			:= F_Read_RegFloat32(PM:= PM, address:=ION9000_E_Voltage_CA);
	PM.Basic.Voltage_LLAvg 			:= F_Read_RegFloat32(PM:= PM, address:=ION9000_E_Voltage_LLAvg);
	PM.Basic.Voltage_AN 			:= F_Read_RegFloat32(PM:= PM, address:=ION9000_E_Voltage_AN);
	PM.Basic.Voltage_BN 			:= F_Read_RegFloat32(PM:= PM, address:=ION9000_E_Voltage_BN);
	PM.Basic.Voltage_CN 			:= F_Read_RegFloat32(PM:= PM, address:=ION9000_E_Voltage_CN);
	PM.Basic.Voltage_LNAvg 			:= F_Read_RegFloat32(PM:= PM, address:=ION9000_E_Voltage_LNAvg);
		
	PM.Basic.Current_A 				:= F_Read_RegFloat32(PM:= PM, address:=ION9000_E_Current_A);
	PM.Basic.Current_B 				:= F_Read_RegFloat32(PM:= PM, address:=ION9000_E_Current_B);
	PM.Basic.Current_C 				:= F_Read_RegFloat32(PM:= PM, address:=ION9000_E_Current_C);
	PM.Basic.Current_N 				:= F_Read_RegFloat32(PM:= PM, address:=ION9000_E_Current_N);
	PM.Basic.Current_G 				:= F_Read_RegFloat32(PM:= PM, address:=ION9000_E_Current_G);
	PM.Basic.Current_Avg 			:= F_Read_RegFloat32(PM:= PM, address:=ION9000_E_Current_Avg);
	
	PM.Basic.RealEnergy_IntoLoad 					:= F_Read_RegInt64(PM:= PM, address:=ION9000_E_RealEnergy_IntoLoad);
	PM.Basic.RealEnergy_OutLoad 					:= F_Read_RegInt64(PM:= PM, address:=ION9000_E_RealEnergy_OutLoad);
	PM.Basic.RealEnergy_Absolute 					:= F_Read_RegInt64(PM:= PM, address:=ION9000_E_RealEnergy_Absolute);
	PM.Basic.RealEnergy_Signed 						:= F_Read_RegInt64(PM:= PM, address:=ION9000_E_RealEnergy_Signed);
	PM.Basic.ReactiveEnergy_IntoLoad 				:= F_Read_RegInt64(PM:= PM, address:=ION9000_E_ReactiveEnergy_IntoLoad);
	PM.Basic.ReactiveEnergy_OutLoad 				:= F_Read_RegInt64(PM:= PM, address:=ION9000_E_ReactiveEnergy_OutLoad);
	PM.Basic.ReactiveEnergy_Absolute 				:= F_Read_RegInt64(PM:= PM, address:=ION9000_E_ReactiveEnergy_Absolute);
	PM.Basic.ReactiveEnergy_Signed 					:= F_Read_RegInt64(PM:= PM, address:=ION9000_E_ReactiveEnergy_Signed);
	PM.Basic.ApparentEnergy_IntoLoad 				:= F_Read_RegInt64(PM:= PM, address:=ION9000_E_ApparentEnergy_IntoLoad);
	PM.Basic.ApparentEnergy_OutLoad 				:= F_Read_RegInt64(PM:= PM, address:=ION9000_E_ApparentEnergy_OutLoad);
	PM.Basic.ApparentEnergy 						:= F_Read_RegInt64(PM:= PM, address:=ION9000_E_ApparentEnergy);
	PM.Basic.ApparentEnergy_Delivered_Received 		:= F_Read_RegInt64(PM:= PM, address:=ION9000_E_ApparentEnergy_Delivered_Received);
	
	PM.Basic.Frequency 				:= F_Read_RegFloat32(PM:= PM, address:=ION9000_E_Frequency );
	PM.Basic.PowerFactor			:= -1*F_Read_RegFloat32(PM := PM, address :=  ION9000_E_PowerFactor);	
	PM.Basic.THDF_Current_A 		:=  100* F_Read_RegFloat32(PM := PM, address := ION9000_E_THDF_Current_A-15000);
	PM.Basic.THDF_Current_B			:= 100* F_Read_RegFloat32(PM := PM, address := ION9000_E_THDF_Current_b-15000);
	PM.Basic.THDF_Current_C 		:= 100* F_Read_RegFloat32(PM := PM, address := ION9000_E_THDF_Current_c-15000);
	PM.Basic.THDF_Current_N 		:= 100* F_Read_RegFloat32(PM := PM, address := ION9000_E_THDF_Current_g-15000);
	PM.Basic.THDF_Voltage_LN		:= 100* F_Read_RegFloat32(PM := PM, address := ION9000_E_THDF_Voltage_LN-15000);
	PM.Basic.THDF_Voltage_AB		:= 100* F_Read_RegFloat32(PM := PM, address := ION9000_E_THDF_Voltage_AN-15000);
	PM.Basic.THDF_Voltage_BC		:= 100* F_Read_RegFloat32(PM := PM, address := ION9000_E_THDF_Voltage_BN-15000);	
	PM.Basic.THDF_Voltage_CA		:= 100* F_Read_RegFloat32(PM := PM, address := ION9000_E_THDF_Voltage_CN-15000);
	nState		:=	STATE_IDLE;	
	nMBAddr		:= 	0;
	Q			:= 	FALSE;
	bDoReading	:= 	FALSE;

	(*PM.Basic.RealEnergy_IntoLoad := F_RoundLrealEx(	lrIn 	:= PM.Basic.RealEnergy_IntoLoad,
										iPrecision 	:= 0);*)
												
	PM.Basic.PowerFactor := F_RoundLrealEx(	lrIn 	:= PM.Basic.PowerFactor,
								iPrecision 	:= 2);
								
	IF IsGoodData (pm.Basic.RealEnergy_IntoLoad )  THEN
		;// pm.Basic.RealEnergy_IntoLoad still it
		validEnvergyIntoLoad := pm.Basic.RealEnergy_IntoLoad;
	ELSE
		pm.Basic.RealEnergy_IntoLoad := validEnvergyIntoLoad;
	END_IF	
								
END_CASE

END_FUNCTION_BLOCK

// ---- POUs/Program/IP237.TcPOU
PROGRAM IP237
VAR
	
	timer				: TON;
	nState				: INT := STATE_INIT;
	
	fbInit237_01_5500			: FB_InitPM;
	fbInit237_02_5500			: FB_InitPM;
	fbInit237_03_5500			: FB_InitPM;
	fbInit237_04_5500			: FB_InitPM;
	fbInit237_05_5500			: FB_InitPM;
	
	fbRead237_01_5500			: FB_PM_ION_9000;
	fbRead237_02_5500			: FB_PM_ION_9000;
	
	//Update 29-08-2022
	fbRead237_03_5500			: FB_ReadPM5350;
	
	//Update 29-08-2022
	fbRead237_04_5500			: FB_ReadPM5350;
	
	//Update 29-08-2022
	fbRead237_05_5500			: FB_ReadPM5350;
	
	
	ipAddr						: STRING := '10.91.37.237';
	nCount						: DINT;
	nQuantity					: WORD:=125;
	nMBAddr						: WORD:=1;
	bExec						: BOOL;
	bBusy						: BOOL;
	bError						: BOOL;
	nErrorId					:UDINT;
	cbRead						: UDINT;
	bOnTest						:bool;
	PMRawDataTest				:ST_PowerMeter;
	// UPDATE BY SUN
	fbInit237_06_5350			: FB_InitPM;
	fbInit237_07_5350			: FB_InitPM;
	fbInit237_08_5350			: FB_InitPM;
	fbInit237_09_5350			: FB_InitPM;
	fbInit237_10_5350			: FB_InitPM;
	fbInit237_11_5350			: FB_InitPM;
	fbInit237_12_5350			: FB_InitPM;
	fbInit237_13_5350			: FB_InitPM;
	
	fbRead237_06_5350			: FB_ReadPM5350;
	fbRead237_07_5350			: FB_ReadPM5350;
	fbRead237_08_5350			: FB_ReadPM5350;
	fbRead237_09_5350			: FB_ReadPM5350;
	fbRead237_10_5350			: FB_ReadPM5350;
	fbRead237_11_5350			: FB_ReadPM5350;
	fbRead237_12_5350			: FB_ReadPM5350;
	fbRead237_13_5350			: FB_ReadPM5350;
	
END_VAR

VAR CONSTANT
	STATE_INIT			:	INT		:= 0;
	STATE_WAIT_CMD		: 	INT		:= 5;
	STATE_READ1			:	INT		:= 10;
	STATE_READ2			:	INT		:= 20;
	STATE_READ3			:	INT		:= 30;
	STATE_READ4			:	INT		:= 40;
	STATE_READ5			:	INT		:= 50;
	////////////////////////////////////////
	STATE_READ6 		:	INT		:= 60;
	STATE_READ7			:	INT		:= 70;
	STATE_READ8			:	INT		:= 80;
	STATE_READ9			:	INT		:= 90;
	STATE_READ10		:	INT		:= 100;
	STATE_READ11		:	INT		:= 110;
	STATE_READ12		:	INT		:= 120;
	STATE_READ13		:	INT		:= 130;
		

END_VAR

CASE nState OF
	STATE_INIT:
		fbInit237_01_5500(	sIpAddress	:= '10.91.37.227',
							nPort		:= 502,
							nUnitID		:= 255,
							PM			:= pmDev.DB07_01_5500);
		fbInit237_02_5500(	sIpAddress	:= '10.91.37.228',
							nPort		:= 502,
							nUnitID		:= 255,
							PM			:= pmDev.DB07_02_5500);
		fbInit237_03_5500(	sIpAddress	:= '10.91.37.237',
							nPort		:= 502,
							nUnitID		:= 3,
							PM			:= pmDev.DB07_03_5500);
		fbInit237_04_5500(	sIpAddress	:= '10.91.37.237',
							nPort		:= 502,
							nUnitID		:= 4,
							PM			:= pmDev.DB07_04_5500);
		fbInit237_05_5500(	sIpAddress	:= '10.91.37.237',
							nPort		:= 502,
							nUnitID		:= 5,
							PM			:= pmDev.DB07_05_5500);
		// updata by sun///////////////////////////////////////////////
		
		fbInit237_06_5350(	sIpAddress	:= '10.91.37.237',
							nPort		:= 502,
							nUnitID		:= 6,
							PM			:= pmDev.DB07_06_5350);
							
		fbInit237_07_5350(	sIpAddress	:= '10.91.37.237',
							nPort		:= 502,
							nUnitID		:= 7,
							PM			:= pmDev.DB07_07_5350);
							
		fbInit237_08_5350(	sIpAddress	:= '10.91.37.237',
							nPort		:= 502,
							nUnitID		:= 8,
							PM			:= pmDev.DB07_08_5350);
							
		fbInit237_09_5350(	sIpAddress	:= '10.91.37.237',
							nPort		:= 502,
							nUnitID		:= 9,
							PM			:= pmDev.DB07_09_5350);
							
		fbInit237_10_5350(	sIpAddress	:= '10.91.37.237',
							nPort		:= 502,
							nUnitID		:= 10,
							PM			:= pmDev.DB07_10_5350);
							
		fbInit237_11_5350(	sIpAddress	:= '10.91.37.237',
							nPort		:= 502,
							nUnitID		:= 11,
							PM			:= pmDev.DB07_11_5350);
							
		fbInit237_12_5350(	sIpAddress	:= '10.91.37.237',
							nPort		:= 502,
							nUnitID		:= 12,
							PM			:= pmDev.DB07_12_5350);
							
		fbInit237_13_5350(	sIpAddress	:= '10.91.37.237',
							nPort		:= 502,
							nUnitID		:= 13,
							PM			:= pmDev.DB07_13_5350);
							
		timer(In:=TRUE, PT:= TIME_INIT);
		IF timer.Q THEN
			timer(In:=FALSE);
			nState	:= STATE_WAIT_CMD;
		END_IF
			
	STATE_WAIT_CMD:
			;
			
	STATE_READ1:
		fbRead237_01_5500(
			bExecute:=TRUE,
			PM:= pmDev.DB07_01_5500);
		IF NOT fbRead237_01_5500.Q THEN
			nState	:= STATE_READ2;
			fbRead237_01_5500(
				bExecute:=FALSE,
				PM:= pmDev.DB07_01_5500);
		END_IF
		
	STATE_READ2:
		fbRead237_02_5500(
			bExecute:=TRUE,
			PM:= pmDev.DB07_02_5500);
		IF NOT fbRead237_02_5500.Q THEN
			nState	:= STATE_READ3;
			fbRead237_02_5500(
				bExecute:=FALSE,
				PM:= pmDev.DB07_02_5500);
		END_IF	
	
	STATE_READ3:
	
		
		fbRead237_03_5500(
			bExecute:=TRUE,
			PM:= pmDev.DB07_03_5500);
		IF NOT fbRead237_03_5500.Q THEN
			nState	:= STATE_READ4;
			fbRead237_03_5500(
				bExecute:=FALSE,
				PM:= pmDev.DB07_03_5500);
		END_IF	
		
	STATE_READ4:
	
		
		fbRead237_04_5500(
			bExecute:=TRUE,
			PM:= pmDev.DB07_04_5500);
		IF NOT fbRead237_04_5500.Q THEN
			nState	:= STATE_READ5;
			fbRead237_04_5500(
				bExecute:=FALSE,
				PM:= pmDev.DB07_04_5500);
		END_IF
		
	STATE_READ5:
	
	
		fbRead237_05_5500(
			bExecute:=TRUE,
			PM:= pmDev.DB07_05_5500);
		IF NOT fbRead237_05_5500.Q THEN
			nState	:= STATE_READ6;
			fbRead237_05_5500(
				bExecute:=FALSE,
				PM:= pmDev.DB07_05_5500);
		END_IF
	
		////////////////////////////update by Sun
		
	STATE_READ6:
	
		fbRead237_06_5350(
			bExecute:=TRUE,
			PM:= pmDev.DB07_06_5350);
		IF NOT fbRead237_06_5350.Q THEN
			nState	:= STATE_READ7;
			fbRead237_06_5350(
				bExecute:=FALSE,
				PM:= pmDev.DB07_06_5350);
		END_IF
	
	STATE_READ7:
	
		fbRead237_07_5350(
			bExecute:=TRUE,
			PM:= pmDev.DB07_07_5350);
		IF NOT fbRead237_07_5350.Q THEN
			nState	:= STATE_READ8;
			fbRead237_07_5350(
				bExecute:=FALSE,
				PM:= pmDev.DB07_07_5350);
		END_IF
	
	STATE_READ8:
	
		fbRead237_08_5350(
			bExecute:=TRUE,
			PM:= pmDev.DB07_08_5350);
		IF NOT fbRead237_08_5350.Q THEN
			nState	:= STATE_READ9;
			fbRead237_08_5350(
				bExecute:=FALSE,
				PM:= pmDev.DB07_08_5350);
		END_IF
	
	STATE_READ9:
	
		fbRead237_09_5350(
			bExecute:=TRUE,
			PM:= pmDev.DB07_09_5350);
		IF NOT fbRead237_09_5350.Q THEN
			nState	:= STATE_READ10;
			fbRead237_09_5350(
				bExecute:=FALSE,
				PM:= pmDev.DB07_09_5350);
		END_IF
		
	STATE_READ10:
	
		fbRead237_10_5350(
			bExecute:=TRUE,
			PM:= pmDev.DB07_10_5350);
		IF NOT fbRead237_10_5350.Q THEN
			nState	:= STATE_READ11;
			fbRead237_10_5350(
				bExecute:=FALSE,
				PM:= pmDev.DB07_10_5350);
		END_IF
	
	STATE_READ11:
	
		fbRead237_11_5350(
			bExecute:=TRUE,
			PM:= pmDev.DB07_11_5350);
		IF NOT fbRead237_11_5350.Q THEN
			nState	:= STATE_READ12;
			fbRead237_11_5350(
				bExecute:=FALSE,
				PM:= pmDev.DB07_11_5350);
		END_IF
	
	STATE_READ12:
	
		fbRead237_12_5350(
			bExecute:=TRUE,
			PM:= pmDev.DB07_12_5350);
		IF NOT fbRead237_12_5350.Q THEN
			nState	:= STATE_READ13;
			fbRead237_12_5350(
				bExecute:=FALSE,
				PM:= pmDev.DB07_12_5350);
		END_IF
	
	STATE_READ13:
	
		fbRead237_13_5350(
			bExecute:=TRUE,
			PM:= pmDev.DB07_13_5350);
		IF NOT fbRead237_13_5350.Q THEN
			nState	:= STATE_WAIT_CMD;
			fbRead237_13_5350(
				bExecute:=FALSE,
				PM:= pmDev.DB07_13_5350);
		END_IF
	

	
END_CASE

PROPERTY Busy : Bool
GET
Busy := nState <> STATE_WAIT_CMD;
END_GET
END_PROPERTY

METHOD Mr_Read : BOOL
VAR_INPUT
END_VAR
IF nState = STATE_WAIT_CMD THEN
	nState := STATE_READ1;
END_IF
END_METHOD

END_PROGRAM

// ---- POUs/Platform/PRG_MachineLogger.TcPOU
PROGRAM PRG_MachineLogger
VAR CONSTANT
	sMACHINE_LOGGER_NAME		: STRING := 'PMS';
	sMACHINE_LOGGER_DIRECTORY	: STRING := '\Hard Disk\';
	sMACHINE_LOGGER_FILE_NAME	: STRING := 'Machine_Logger_';
END_VAR
VAR
	bFirstCycle : BOOL	:= TRUE; (* Auxilary bit for initial setup assignaments *)
	bTestWrite : BOOL;
	bActivated : BOOL; 
END_VAR

IF bFirstCycle THEN
	bFirstCycle := FALSE;
	fbMachineLogger.MR_FirstCycle(	sName 			:= sMACHINE_LOGGER_NAME,
									sFileDir		:= sMACHINE_LOGGER_DIRECTORY,
									sFileName 		:= sMACHINE_LOGGER_FILE_NAME,
									sAmsNetId 		:= '',
									bAddTimeStamp	:= TRUE,
									bAddHeader		:= TRUE);

	

END_IF

IF NOT fbMachineLogger.Active THEN
	fbMachineLogger.MR_Init();
END_IF
(* Cyclic run *)
fbMachineLogger();
IF bTestWrite THEN
	bTestWrite := 0;
	fbMachineLogger.MR_AddLogs( sLogMessage := 'this is test add log');
END_IF

END_PROGRAM

// ---- POUs/Program/PmReport2.TcPOU
PROGRAM PmReport2
VAR
	arCalculateEnergy_1H : ARRAY [0..pmDev.numAllMeter-1] OF FB_CalCulateAccumulation;
	arFIFOEnergy_1H		 : ARRAY [0..pmDev.numAllMeter-1] OF FB_FIFO_Lreal;
	arCalculateEnergy_1D : ARRAY [0..pmDev.numAllMeter-1] OF FB_CalCulateAccumulation;
	arFIFOEnergy_1D 	 : ARRAY [0..pmDev.numAllMeter-1] OF FB_FIFO_Lreal;
	FIFOEnergyTimestruct_1H :  FB_FIFO_TimeStruct;
	FIFOEnergyTimestruct_1D :  FB_FIFO_TimeStruct;
	AllInitSuccessful : BOOL := TRUE;
	iloop  : UINT;
	eState	: UINT;
	tonPrepareValue: TON;
	tTimePrepareValue: TIME := t#2S;
END_VAR
VAR CONSTANT
	STATE_INIT 							: UINT := 0;
	STATE_RUN							: UINT := 10;
	STATE_REPORT_WAIT 					: UINT := 0;
	STATE_REPORT_ENERGY_HOUR_REQUEST 	: UINT := 10;
	STATE_REPORT_ENERGY_HOUR_ACTIVE_REQUEST	:UINT := 15;
	STATE_REPORT_ENERGY_HOUR_WAIT_ACK		: UINT := 20;
	
	STATE_REPORT_ENERGY_DAY_REQUEST 	: UINT := 50;
	STATE_REPORT_ENERGY_DAY_ACTIVE_REQUEST	:UINT := 55;
	STATE_REPORT_ENERGY_DAY_WAIT_ACK			: UINT := 60;
END_VAR
VAR PERSISTENT 
	
	eStateReport : UINT;
	bEnergyReportHourEvent : BOOL;// is true if IPC request Report Energy HOUR to AVEVA, FALSE if AVEVA Ack processed The data
	bEnergyReportDayEvent : BOOL;// is true if IPC request Report Energy DAY to AVEVA, FALSE if AVEVA Ack processed The data
	sDateAndTimeReportAveva : STRING;
	sMsReportAveva			: STRING;
	
	// virtual object
	////Power Virtual Meter	// new require 19/07	
		MaySayKhi			: 	LREAL;
		OilCoolingPump		: 	LREAL;
		LightNVO			: 	LREAL;
		CP_WHEF1            : 	LREAL;
		CP_WHEF2            :	LREAL;
		DB_FIC              :	LREAL;
	
	// date 2508
	//Machine
		PKG_HoongA			: 	LREAL;
		PKG_Other			: 	LREAL;
		TE_Tufting			: 	LREAL;
		TE_End				:	LREAL;
		IM_VIM				: 	LREAL;
		IM_HIM				: 	LREAL;
		MIXING				: 	LREAL;
		LIGHTING_IM			: 	LREAL;
		LIGHTING_PKG_TE		: 	LREAL;
		AIRCOMP1       : LREAL;
		AIRCOMP2       : LREAL;
		AIRCOMP3       : LREAL;
		AIRCOMP4       : LREAL;
		AIRCOMP5       : LREAL;
		BLISTER_FORMING       : LREAL;
		LIGHTING_BLISTER       : LREAL;
		CHILLER4       : LREAL;
		CHILLER5       : LREAL;
		CHILLER6       : LREAL;
		OIL_COOLING       : LREAL;
		TE_AFT       : LREAL;
		TE_HEPTA       : LREAL;
		TE_FREXILINE       : LREAL;
		OFFICE_GROUND       : LREAL;
		OFFICE_1       : LREAL;
		CANTEEN       : LREAL;
		SECURITY_FONT       : LREAL;
		SECURITY_BACK       : LREAL;
		LIGHTING_RM       : LREAL;
		LIGHTING_FG       : LREAL;
	//Area
		PKG       : LREAL;
		TE       : LREAL;
		IM       : LREAL;
		AreaMixing       : LREAL;
		Lighting       : LREAL;
		Aircomp       : LREAL;
		HVACAHU       : LREAL;
		GROUND       : LREAL;
		Layer1       : LREAL;
		HVAC       : LREAL;
		Kit        : LREAL;
		Chiller       : LREAL;
		Other       : LREAL;
		
		//Hour
		// virtual object
	////Power Virtual Meter	// new require 19/07	
		MaySayKhi_H			: 	LREAL;
		OilCoolingPump_H		: 	LREAL;
		LightNVO_H				: 	LREAL;
		CP_WHEF1_H	            : 	LREAL;
		CP_WHEF2_H	            :	LREAL;
		DB_FIC_H	              :	LREAL;
	
	// date 2508
	//Machine
		PKG_HoongA_H				: 	LREAL;
		PKG_Other_H				: 	LREAL;
		TE_Tufting_H				: 	LREAL;
		TE_End_H					:	LREAL;
		IM_VIM_H					: 	LREAL;
		IM_HIM_H					: 	LREAL;
		MIXING_H					: 	LREAL;
		LIGHTING_IM_H				: 	LREAL;
		LIGHTING_PKG_TE_H			: 	LREAL;
		AIRCOMP1_H	       : LREAL;
		AIRCOMP2_H	       : LREAL;
		AIRCOMP3_H	       : LREAL;
		AIRCOMP4_H	       : LREAL;
		AIRCOMP5_H	       : LREAL;
		BLISTER_FORMING_H	       : LREAL;
		LIGHTING_BLISTER_H	       : LREAL;
		CHILLER4_H	       : LREAL;
		CHILLER5_H	       : LREAL;
		CHILLER6_H	       : LREAL;
		OIL_COOLING_H	       : LREAL;
		TE_AFT_H	       : LREAL;
		TE_HEPTA_H	       : LREAL;
		TE_FREXILINE_H	       : LREAL;
		OFFICE_GROUND_H	       : LREAL;
		OFFICE_1_H	       : LREAL;
		CANTEEN_H	       : LREAL;
		SECURITY_FONT_H	       : LREAL;
		SECURITY_BACK_H	       : LREAL;
		LIGHTING_RM_H	       : LREAL;
		LIGHTING_FG_H	       : LREAL;
	//Area
		PKG_H	       : LREAL;
		TE_H	       : LREAL;
		IM_H	       : LREAL;
		AreaMixing_H	       : LREAL;
		Lighting_H	       : LREAL;
		Aircomp_H	       : LREAL;
		HVACAHU_H	       : LREAL;
		GROUND_H	       : LREAL;
		Layer1_H	       : LREAL;
		HVAC_H	       : LREAL;
		Kit_H	        : LREAL;
		Chiller_H	       : LREAL;
		Other_H	       : LREAL;
END_VAR



CASE eState OF
	STATE_INIT:
		Init();
	STATE_RUN:
		Run();
	;
	
END_CASE

METHOD CalculateVirtualObject : BOOL
VAR_INPUT
END_VAR
///require 25/08	
	//Area
		PKG   :=	arFIFOEnergy_1D[ DB1].OldestData
												+arFIFOEnergy_1D[ DB2].OldestData
												+arFIFOEnergy_1D[ DB11].OldestData ;
												
		TE    := arFIFOEnergy_1D[ DB3].OldestData
												+arFIFOEnergy_1D[ DB10].OldestData
												+arFIFOEnergy_1D[ DB12].OldestData;
												
		IM    := arFIFOEnergy_1D[ DB4].OldestData
												+arFIFOEnergy_1D[ DB5].OldestData
												+arFIFOEnergy_1D[ DB6].OldestData
												+arFIFOEnergy_1D[ DB7].OldestData
												+arFIFOEnergy_1D[ DB8].OldestData
												+arFIFOEnergy_1D[ DB9].OldestData;
												
		AreaMixing   := arFIFOEnergy_1D[ DB_MR].OldestData;
		Lighting     := arFIFOEnergy_1D[ LP_PR1A].OldestData
														+arFIFOEnergy_1D[ LP_PR1B].OldestData
														+arFIFOEnergy_1D[ LP_PR2A].OldestData
														+arFIFOEnergy_1D[ LP_PR2B].OldestData
														+arFIFOEnergy_1D[ LP_PR3A].OldestData
														+arFIFOEnergy_1D[ LP_PR3B].OldestData
														+arFIFOEnergy_1D[ LP_PR4A].OldestData
														+arFIFOEnergy_1D[ LP_PR4B].OldestData
														+arFIFOEnergy_1D[ LP_BM].OldestData
														+arFIFOEnergy_1D[ LP_WH1].OldestData
														+arFIFOEnergy_1D[ LP_WH2].OldestData
														+arFIFOEnergy_1D[ LP_PR5A].OldestData
														+arFIFOEnergy_1D[ LP_PR5B].OldestData
														+arFIFOEnergy_1D[ LP_PR6A].OldestData
														+arFIFOEnergy_1D[ LP_PR6B].OldestData;
														
		Aircomp   := arFIFOEnergy_1D[ DB_AIRCOMP].OldestData;
		HVACAHU   := arFIFOEnergy_1D[ DB_AHU].OldestData;
		GROUND    := arFIFOEnergy_1D[ DB_OFF1].OldestData;
		Layer1    := arFIFOEnergy_1D[ DB_OFF2].OldestData;
		HVAC      := arFIFOEnergy_1D[ DB_MVAC1].OldestData;
		Kit       := arFIFOEnergy_1D[ DB_kit].OldestData;
		Chiller   := arFIFOEnergy_1D[ DB_MVAC2].OldestData;
		Other     := arFIFOEnergy_1D[ LV01].OldestData
														+arFIFOEnergy_1D[ LV02].OldestData
														+arFIFOEnergy_1D[ LV03].OldestData
														+arFIFOEnergy_1D[ LV04].OldestData;
	//Machine
		PKG_HoongA         :=    arFIFOEnergy_1D[ DB1_1].OldestData
																+arFIFOEnergy_1D[ DB2_1].OldestData
																+arFIFOEnergy_1D[ DB11_1].OldestData;
																		
		PKG_Other      :=   arFIFOEnergy_1D[ DB1_2].OldestData
																+arFIFOEnergy_1D[ DB2_2].OldestData
																+arFIFOEnergy_1D[ DB11_2].OldestData;
		TE_Tufting     :=   arFIFOEnergy_1D[ DB3_1].OldestData
																+arFIFOEnergy_1D[ DB10_1].OldestData
																+arFIFOEnergy_1D[ DB12_1].OldestData;
		TE_End         :=   arFIFOEnergy_1D[ DB3_2].OldestData
																+arFIFOEnergy_1D[ DB10_2].OldestData
																+arFIFOEnergy_1D[ DB12_2].OldestData;
		IM_VIM         :=   arFIFOEnergy_1D[ DB4_1].OldestData
																+arFIFOEnergy_1D[ DB5_1].OldestData
																+arFIFOEnergy_1D[ DB6_1].OldestData
																+arFIFOEnergy_1D[ DB7_1].OldestData
																+arFIFOEnergy_1D[ DB8_1].OldestData
																+arFIFOEnergy_1D[ DB9_1].OldestData;
		IM_HIM         :=    arFIFOEnergy_1D[ DB4_2].OldestData
																+arFIFOEnergy_1D[ DB5_2].OldestData
																+arFIFOEnergy_1D[ DB6_2].OldestData
																+arFIFOEnergy_1D[ DB7_2].OldestData
																+arFIFOEnergy_1D[ DB8_2].OldestData
																+arFIFOEnergy_1D[ DB9_2].OldestData
																+arFIFOEnergy_1D[ DB14_2].OldestData
																+arFIFOEnergy_1D[ DB15_2].OldestData
																+arFIFOEnergy_1D[ DB13_2].OldestData;
																
		MIXING         :=    arFIFOEnergy_1D[ DB_MR].OldestData;
		LIGHTING_IM    :=    arFIFOEnergy_1D[ LP_PR1A].OldestData
																+arFIFOEnergy_1D[ LP_PR1B].OldestData
																+arFIFOEnergy_1D[ LP_PR3A].OldestData
																+arFIFOEnergy_1D[ LP_PR3B].OldestData
																+arFIFOEnergy_1D[ LP_PR5A].OldestData
																+arFIFOEnergy_1D[ LP_PR5B].OldestData;
																
		LIGHTING_PKG_TE  :=  arFIFOEnergy_1D[ LP_PR4A].OldestData
																+arFIFOEnergy_1D[ LP_PR4B].OldestData
																+arFIFOEnergy_1D[ LP_PR2A].OldestData
																+arFIFOEnergy_1D[ LP_PR2B].OldestData
																+arFIFOEnergy_1D[ LP_PR6A].OldestData
																+arFIFOEnergy_1D[ LP_PR6B].OldestData;
																
		AIRCOMP1         :=          arFIFOEnergy_1D[ A1].OldestData;
		AIRCOMP2         :=          arFIFOEnergy_1D[ A2].OldestData;
		AIRCOMP3         :=          arFIFOEnergy_1D[ A3].OldestData;
		AIRCOMP4         :=          arFIFOEnergy_1D[ A4].OldestData;
		AIRCOMP5         :=          arFIFOEnergy_1D[ A5].OldestData;
		BLISTER_FORMING         :=          arFIFOEnergy_1D[ DB_BM].OldestData;
		LIGHTING_BLISTER         :=          arFIFOEnergy_1D[ LP_BM].OldestData;
		CHILLER4         :=          arFIFOEnergy_1D[ CH4].OldestData;
		CHILLER5         :=          arFIFOEnergy_1D[ CH5].OldestData;
		CHILLER6         :=          arFIFOEnergy_1D[ CH6].OldestData;
		OIL_COOLING         :=          arFIFOEnergy_1D[ DB_MVAC1].OldestData;
		TE_AFT         :=          arFIFOEnergy_1D[ DB13_1].OldestData;
		TE_HEPTA         :=          arFIFOEnergy_1D[ DB14_1].OldestData;
		TE_FREXILINE         :=          arFIFOEnergy_1D[ DB15_1].OldestData;
		OFFICE_GROUND         :=          arFIFOEnergy_1D[ DB_OFF1].OldestData;
		OFFICE_1         :=          arFIFOEnergy_1D[ DB_OFF2].OldestData;
		CANTEEN         :=          arFIFOEnergy_1D[ DB_KIT].OldestData;
		SECURITY_FONT         :=          arFIFOEnergy_1D[ LP_EL1].OldestData;
		SECURITY_BACK         :=          arFIFOEnergy_1D[ LP_EL2].OldestData;
		LIGHTING_RM         :=          arFIFOEnergy_1D[ LP_WH1].OldestData;
		LIGHTING_FG         :=          arFIFOEnergy_1D[ LP_WH2].OldestData;
//hour
///require 25/08	
	//Area
		PKG_H	   :=	arFIFOEnergy_1H[ DB1].OldestData
												+arFIFOEnergy_1H[ DB2].OldestData
												+arFIFOEnergy_1H[ DB11].OldestData ;
												
		TE_H	    := arFIFOEnergy_1H[ DB3].OldestData
												+arFIFOEnergy_1H[ DB10].OldestData
												+arFIFOEnergy_1H[ DB12].OldestData;
												
		IM_H	    := arFIFOEnergy_1H[ DB4].OldestData
												+arFIFOEnergy_1H[ DB5].OldestData
												+arFIFOEnergy_1H[ DB6].OldestData
												+arFIFOEnergy_1H[ DB7].OldestData
												+arFIFOEnergy_1H[ DB8].OldestData
												+arFIFOEnergy_1H[ DB9].OldestData;
												
		AreaMixing_H	   := arFIFOEnergy_1H[ DB_MR].OldestData;
		Lighting_H	     := arFIFOEnergy_1H[ LP_PR1A].OldestData
														+arFIFOEnergy_1H[ LP_PR1B].OldestData
														+arFIFOEnergy_1H[ LP_PR2A].OldestData
														+arFIFOEnergy_1H[ LP_PR2B].OldestData
														+arFIFOEnergy_1H[ LP_PR3A].OldestData
														+arFIFOEnergy_1H[ LP_PR3B].OldestData
														+arFIFOEnergy_1H[ LP_PR4A].OldestData
														+arFIFOEnergy_1H[ LP_PR4B].OldestData
														+arFIFOEnergy_1H[ LP_BM].OldestData
														+arFIFOEnergy_1H[ LP_WH1].OldestData
														+arFIFOEnergy_1H[ LP_WH2].OldestData
														+arFIFOEnergy_1H[ LP_PR5A].OldestData
														+arFIFOEnergy_1H[ LP_PR5B].OldestData
														+arFIFOEnergy_1H[ LP_PR6A].OldestData
														+arFIFOEnergy_1H[ LP_PR6B].OldestData;
														
		Aircomp_H	   := arFIFOEnergy_1H[ DB_AIRCOMP].OldestData;
		HVACAHU_H	   := arFIFOEnergy_1H[ DB_AHU].OldestData;
		GROUND_H	    := arFIFOEnergy_1H[ DB_OFF1].OldestData;
		Layer1_H	    := arFIFOEnergy_1H[ DB_OFF2].OldestData;
		HVAC_H	      := arFIFOEnergy_1H[ DB_MVAC1].OldestData;
		Kit_H	       := arFIFOEnergy_1H[ DB_kit].OldestData;
		Chiller_H	   := arFIFOEnergy_1H[ DB_MVAC2].OldestData;
		Other_H	     := arFIFOEnergy_1H[ LV01].OldestData
														+arFIFOEnergy_1H[ LV02].OldestData
														+arFIFOEnergy_1H[ LV03].OldestData
														+arFIFOEnergy_1H[ LV04].OldestData;
	//Machine
		PKG_HoongA_H	         :=    arFIFOEnergy_1H[ DB1_1].OldestData
																+arFIFOEnergy_1H[ DB2_1].OldestData
																+arFIFOEnergy_1H[ DB11_1].OldestData;
																		
		PKG_Other_H	      :=   arFIFOEnergy_1H[ DB1_2].OldestData
																+arFIFOEnergy_1H[ DB2_2].OldestData
																+arFIFOEnergy_1H[ DB11_2].OldestData;
		TE_Tufting_H	     :=   arFIFOEnergy_1H[ DB3_1].OldestData
																+arFIFOEnergy_1H[ DB10_1].OldestData
																+arFIFOEnergy_1H[ DB12_1].OldestData;
		TE_End_H	         :=   arFIFOEnergy_1H[ DB3_2].OldestData
																+arFIFOEnergy_1H[ DB10_2].OldestData
																+arFIFOEnergy_1H[ DB12_2].OldestData;
		IM_VIM_H	         :=   arFIFOEnergy_1H[ DB4_1].OldestData
																+arFIFOEnergy_1H[ DB5_1].OldestData
																+arFIFOEnergy_1H[ DB6_1].OldestData
																+arFIFOEnergy_1H[ DB7_1].OldestData
																+arFIFOEnergy_1H[ DB8_1].OldestData
																+arFIFOEnergy_1H[ DB9_1].OldestData;
		IM_HIM_H	         :=    arFIFOEnergy_1H[ DB4_2].OldestData
																+arFIFOEnergy_1H[ DB5_2].OldestData
																+arFIFOEnergy_1H[ DB6_2].OldestData
																+arFIFOEnergy_1H[ DB7_2].OldestData
																+arFIFOEnergy_1H[ DB8_2].OldestData
																+arFIFOEnergy_1H[ DB9_2].OldestData
																+arFIFOEnergy_1H[ DB14_2].OldestData
																+arFIFOEnergy_1H[ DB15_2].OldestData
																+arFIFOEnergy_1H[ DB13_2].OldestData;
																
		MIXING_H	         :=    arFIFOEnergy_1H[ DB_MR].OldestData;
		LIGHTING_IM_H	    :=    arFIFOEnergy_1H[ LP_PR1A].OldestData
																+arFIFOEnergy_1H[ LP_PR1B].OldestData
																+arFIFOEnergy_1H[ LP_PR3A].OldestData
																+arFIFOEnergy_1H[ LP_PR3B].OldestData
																+arFIFOEnergy_1H[ LP_PR5A].OldestData
																+arFIFOEnergy_1H[ LP_PR5B].OldestData;
																
		LIGHTING_PKG_TE_H	  :=  arFIFOEnergy_1H[ LP_PR4A].OldestData
																+arFIFOEnergy_1H[ LP_PR4B].OldestData
																+arFIFOEnergy_1H[ LP_PR2A].OldestData
																+arFIFOEnergy_1H[ LP_PR2B].OldestData
																+arFIFOEnergy_1H[ LP_PR6A].OldestData
																+arFIFOEnergy_1H[ LP_PR6B].OldestData;
																
		AIRCOMP1_H	         :=          arFIFOEnergy_1H[ A1].OldestData;
		AIRCOMP2_H	         :=          arFIFOEnergy_1H[ A2].OldestData;
		AIRCOMP3_H	         :=          arFIFOEnergy_1H[ A3].OldestData;
		AIRCOMP4_H	         :=          arFIFOEnergy_1H[ A4].OldestData;
		AIRCOMP5_H	         :=          arFIFOEnergy_1H[ A5].OldestData;
		BLISTER_FORMING_H	         :=          arFIFOEnergy_1H[ DB_BM].OldestData;
		LIGHTING_BLISTER_H	         :=          arFIFOEnergy_1H[ LP_BM].OldestData;
		CHILLER4_H	         :=          arFIFOEnergy_1H[ CH4].OldestData;
		CHILLER5_H	         :=          arFIFOEnergy_1H[ CH5].OldestData;
		CHILLER6_H	         :=          arFIFOEnergy_1H[ CH6].OldestData;
		OIL_COOLING_H	         :=          arFIFOEnergy_1H[ DB_MVAC1].OldestData;
		TE_AFT_H	         :=          arFIFOEnergy_1H[ DB13_1].OldestData;
		TE_HEPTA_H	         :=          arFIFOEnergy_1H[ DB14_1].OldestData;
		TE_FREXILINE_H	         :=          arFIFOEnergy_1H[ DB15_1].OldestData;
		OFFICE_GROUND_H	         :=          arFIFOEnergy_1H[ DB_OFF1].OldestData;
		OFFICE_1_H	         :=          arFIFOEnergy_1H[ DB_OFF2].OldestData;
		CANTEEN_H	         :=          arFIFOEnergy_1H[ DB_KIT].OldestData;
		SECURITY_FONT_H	         :=          arFIFOEnergy_1H[ LP_EL1].OldestData;
		SECURITY_BACK_H	         :=          arFIFOEnergy_1H[ LP_EL2].OldestData;
		LIGHTING_RM_H	         :=          arFIFOEnergy_1H[ LP_WH1].OldestData;
		LIGHTING_FG_H	         :=          arFIFOEnergy_1H[ LP_WH2].OldestData;
END_METHOD

METHOD Init : BOOL
VAR_INPUT
END_VAR
VAR 
	iloop : UINT;
	
END_VAR
// naming
	//arCalculateEnergy_1H
		arCalculateEnergy_1H[LV01].Name := 'LV01';
		arCalculateEnergy_1H[DB_PR1_1].Name := 'DB_PR1_1';
		arCalculateEnergy_1H[DB1].Name := 'DB1';
		arCalculateEnergy_1H[DB2].Name := 'DB2';
		arCalculateEnergy_1H[DB3].Name := 'DB3';
		arCalculateEnergy_1H[DB4].Name := 'DB4';
		arCalculateEnergy_1H[DB1_1].Name := 'DB1_1';
		arCalculateEnergy_1H[DB2_1].Name := 'DB2_1';
		arCalculateEnergy_1H[DB3_1].Name := 'DB3_1';
		arCalculateEnergy_1H[DB4_1].Name := 'DB4_1';
		arCalculateEnergy_1H[DB5].Name := 'DB5';
		arCalculateEnergy_1H[DB6].Name := 'DB6';
		arCalculateEnergy_1H[DB7].Name := 'DB7';
		arCalculateEnergy_1H[DB_MR].Name := 'DB_MR';
		arCalculateEnergy_1H[DB5_1].Name := 'DB5_1';
		arCalculateEnergy_1H[DB6_1].Name := 'DB6_1';
		arCalculateEnergy_1H[DB7_1].Name := 'DB7_1';
		arCalculateEnergy_1H[LV02].Name := 'LV02';
		arCalculateEnergy_1H[DB_PR1_2].Name := 'DB_PR1_2';
		arCalculateEnergy_1H[DB_AIRCOMP].Name := 'DB_AIRCOMP';
		arCalculateEnergy_1H[DB_AHU].Name := 'DB_AHU';
		arCalculateEnergy_1H[DB8].Name := 'DB8';
		arCalculateEnergy_1H[DB9].Name := 'DB9';
		arCalculateEnergy_1H[DB10].Name := 'DB10';
		arCalculateEnergy_1H[DB8_1].Name := 'DB8_1';
		arCalculateEnergy_1H[DB9_1].Name := 'DB9_1';
		arCalculateEnergy_1H[DB10_1].Name := 'DB10_1';
		arCalculateEnergy_1H[A1].Name := 'A1';
		arCalculateEnergy_1H[A2].Name := 'A2';
		arCalculateEnergy_1H[A3].Name := 'A3';
		arCalculateEnergy_1H[A4].Name := 'A4';
		arCalculateEnergy_1H[A5].Name := 'A5';
		arCalculateEnergy_1H[LP_PR1A].Name := 'LP_PR1A';
		arCalculateEnergy_1H[LP_PR1B].Name := 'LP_PR1B';
		arCalculateEnergy_1H[LP_PR2A].Name := 'LP_PR2A';
		arCalculateEnergy_1H[LP_PR2B].Name := 'LP_PR2B';
		arCalculateEnergy_1H[LP_PR3A].Name := 'LP_PR3A';
		arCalculateEnergy_1H[DB_WH].Name := 'DB_WH';
		arCalculateEnergy_1H[LP_PR3B].Name := 'LP_PR3B';
		arCalculateEnergy_1H[LP_PR4A].Name := 'LP_PR4A';
		arCalculateEnergy_1H[LP_PR4B].Name := 'LP_PR4B';
		arCalculateEnergy_1H[LP_BM].Name := 'LP_BM';
		arCalculateEnergy_1H[DB_BM].Name := 'DB_BM';
		arCalculateEnergy_1H[LV03].Name := 'LV03';
		arCalculateEnergy_1H[DB_MVAC1].Name := 'DB_MVAC1';
		arCalculateEnergy_1H[DB_MVAC2].Name := 'DB_MVAC2';
		arCalculateEnergy_1H[DB_OFF2].Name := 'DB_OFF2';
		arCalculateEnergy_1H[LP_EL1].Name := 'LP_EL1';
		arCalculateEnergy_1H[LP_EL2].Name := 'LP_EL2';
		arCalculateEnergy_1H[DB_OFF1].Name := 'DB_OFF1';
		arCalculateEnergy_1H[DB_KIT].Name := 'DB_KIT';
		arCalculateEnergy_1H[LP_WH2].Name := 'LP_WH2';
		arCalculateEnergy_1H[LP_WH1].Name := 'LP_WH1';
		arCalculateEnergy_1H[CH4].Name := 'CH4';
		arCalculateEnergy_1H[CH5].Name := 'CH5';
		arCalculateEnergy_1H[CH6].Name := 'CH6';
		arCalculateEnergy_1H[LV04].Name := 'LV04';
		arCalculateEnergy_1H[DB_PR2].Name := 'DB_PR2';
		arCalculateEnergy_1H[DB11].Name := 'DB11';
		arCalculateEnergy_1H[DB12].Name := 'DB12';
		arCalculateEnergy_1H[DB13].Name := 'DB13';
		arCalculateEnergy_1H[DB14].Name := 'DB14';
		arCalculateEnergy_1H[DB11_1].Name := 'DB11_1';
		arCalculateEnergy_1H[DB12_1].Name := 'DB12_1';
		arCalculateEnergy_1H[DB13_1].Name := 'DB13_1';
		arCalculateEnergy_1H[DB14_1].Name := 'DB14_1';
		arCalculateEnergy_1H[DB15].Name := 'DB15';
		arCalculateEnergy_1H[DB15_1].Name := 'DB15_1';
		arCalculateEnergy_1H[LP_PR5A].Name := 'LP_PR5A';
		arCalculateEnergy_1H[LP_PR5B].Name := 'LP_PR5B';
		arCalculateEnergy_1H[LP_PR6A].Name := 'LP_PR6A';
		arCalculateEnergy_1H[LP_PR6B].Name := 'LP_PR6B';
		arCalculateEnergy_1H[DB1_2].Name := 'DB1_2';
		arCalculateEnergy_1H[DB2_2].Name := 'DB2_2';
		arCalculateEnergy_1H[DB3_2].Name := 'DB3_2';
		arCalculateEnergy_1H[DB4_2].Name := 'DB4_2';
		arCalculateEnergy_1H[DB5_2].Name := 'DB5_2';
		arCalculateEnergy_1H[DB6_2].Name := 'DB6_2';
		arCalculateEnergy_1H[DB7_2].Name := 'DB7_2';
		arCalculateEnergy_1H[DB8_2].Name := 'DB8_2';
		arCalculateEnergy_1H[DB9_2].Name := 'DB9_2';
		arCalculateEnergy_1H[DB10_2].Name := 'DB10_2';
		arCalculateEnergy_1H[DB11_2].Name := 'DB11_2';
		arCalculateEnergy_1H[DB12_2].Name := 'DB12_2';
		arCalculateEnergy_1H[DB13_2].Name := 'DB13_2';
		arCalculateEnergy_1H[DB14_2].Name := 'DB14_2';
		arCalculateEnergy_1H[DB15_2].Name := 'DB15_2';
		
	//arCalculateEnergy_1D
		arCalculateEnergy_1D[LV01].Name := 'LV01';
		arCalculateEnergy_1D[DB_PR1_1].Name := 'DB_PR1_1';
		arCalculateEnergy_1D[DB1].Name := 'DB1';
		arCalculateEnergy_1D[DB2].Name := 'DB2';
		arCalculateEnergy_1D[DB3].Name := 'DB3';
		arCalculateEnergy_1D[DB4].Name := 'DB4';
		arCalculateEnergy_1D[DB1_1].Name := 'DB1_1';
		arCalculateEnergy_1D[DB2_1].Name := 'DB2_1';
		arCalculateEnergy_1D[DB3_1].Name := 'DB3_1';
		arCalculateEnergy_1D[DB4_1].Name := 'DB4_1';
		arCalculateEnergy_1D[DB5].Name := 'DB5';
		arCalculateEnergy_1D[DB6].Name := 'DB6';
		arCalculateEnergy_1D[DB7].Name := 'DB7';
		arCalculateEnergy_1D[DB_MR].Name := 'DB_MR';
		arCalculateEnergy_1D[DB5_1].Name := 'DB5_1';
		arCalculateEnergy_1D[DB6_1].Name := 'DB6_1';
		arCalculateEnergy_1D[DB7_1].Name := 'DB7_1';
		arCalculateEnergy_1D[LV02].Name := 'LV02';
		arCalculateEnergy_1D[DB_PR1_2].Name := 'DB_PR1_2';
		arCalculateEnergy_1D[DB_AIRCOMP].Name := 'DB_AIRCOMP';
		arCalculateEnergy_1D[DB_AHU].Name := 'DB_AHU';
		arCalculateEnergy_1D[DB8].Name := 'DB8';
		arCalculateEnergy_1D[DB9].Name := 'DB9';
		arCalculateEnergy_1D[DB10].Name := 'DB10';
		arCalculateEnergy_1D[DB8_1].Name := 'DB8_1';
		arCalculateEnergy_1D[DB9_1].Name := 'DB9_1';
		arCalculateEnergy_1D[DB10_1].Name := 'DB10_1';
		arCalculateEnergy_1D[A1].Name := 'A1';
		arCalculateEnergy_1D[A2].Name := 'A2';
		arCalculateEnergy_1D[A3].Name := 'A3';
		arCalculateEnergy_1D[A4].Name := 'A4';
		arCalculateEnergy_1D[A5].Name := 'A5';
		arCalculateEnergy_1D[LP_PR1A].Name := 'LP_PR1A';
		arCalculateEnergy_1D[LP_PR1B].Name := 'LP_PR1B';
		arCalculateEnergy_1D[LP_PR2A].Name := 'LP_PR2A';
		arCalculateEnergy_1D[LP_PR2B].Name := 'LP_PR2B';
		arCalculateEnergy_1D[LP_PR3A].Name := 'LP_PR3A';
		arCalculateEnergy_1D[DB_WH].Name := 'DB_WH';
		arCalculateEnergy_1D[LP_PR3B].Name := 'LP_PR3B';
		arCalculateEnergy_1D[LP_PR4A].Name := 'LP_PR4A';
		arCalculateEnergy_1D[LP_PR4B].Name := 'LP_PR4B';
		arCalculateEnergy_1D[LP_BM].Name := 'LP_BM';
		arCalculateEnergy_1D[DB_BM].Name := 'DB_BM';
		arCalculateEnergy_1D[LV03].Name := 'LV03';
		arCalculateEnergy_1D[DB_MVAC1].Name := 'DB_MVAC1';
		arCalculateEnergy_1D[DB_MVAC2].Name := 'DB_MVAC2';
		arCalculateEnergy_1D[DB_OFF2].Name := 'DB_OFF2';
		arCalculateEnergy_1D[LP_EL1].Name := 'LP_EL1';
		arCalculateEnergy_1D[LP_EL2].Name := 'LP_EL2';
		arCalculateEnergy_1D[DB_OFF1].Name := 'DB_OFF1';
		arCalculateEnergy_1D[DB_KIT].Name := 'DB_KIT';
		arCalculateEnergy_1D[LP_WH2].Name := 'LP_WH2';
		arCalculateEnergy_1D[LP_WH1].Name := 'LP_WH1';
		arCalculateEnergy_1D[CH4].Name := 'CH4';
		arCalculateEnergy_1D[CH5].Name := 'CH5';
		arCalculateEnergy_1D[CH6].Name := 'CH6';
		arCalculateEnergy_1D[LV04].Name := 'LV04';
		arCalculateEnergy_1D[DB_PR2].Name := 'DB_PR2';
		arCalculateEnergy_1D[DB11].Name := 'DB11';
		arCalculateEnergy_1D[DB12].Name := 'DB12';
		arCalculateEnergy_1D[DB13].Name := 'DB13';
		arCalculateEnergy_1D[DB14].Name := 'DB14';
		arCalculateEnergy_1D[DB11_1].Name := 'DB11_1';
		arCalculateEnergy_1D[DB12_1].Name := 'DB12_1';
		arCalculateEnergy_1D[DB13_1].Name := 'DB13_1';
		arCalculateEnergy_1D[DB14_1].Name := 'DB14_1';
		arCalculateEnergy_1D[DB15].Name := 'DB15';
		arCalculateEnergy_1D[DB15_1].Name := 'DB15_1';
		arCalculateEnergy_1D[LP_PR5A].Name := 'LP_PR5A';
		arCalculateEnergy_1D[LP_PR5B].Name := 'LP_PR5B';
		arCalculateEnergy_1D[LP_PR6A].Name := 'LP_PR6A';
		arCalculateEnergy_1D[LP_PR6B].Name := 'LP_PR6B';
		arCalculateEnergy_1D[DB1_2].Name := 'DB1_2';
		arCalculateEnergy_1D[DB2_2].Name := 'DB2_2';
		arCalculateEnergy_1D[DB3_2].Name := 'DB3_2';
		arCalculateEnergy_1D[DB4_2].Name := 'DB4_2';
		arCalculateEnergy_1D[DB5_2].Name := 'DB5_2';
		arCalculateEnergy_1D[DB6_2].Name := 'DB6_2';
		arCalculateEnergy_1D[DB7_2].Name := 'DB7_2';
		arCalculateEnergy_1D[DB8_2].Name := 'DB8_2';
		arCalculateEnergy_1D[DB9_2].Name := 'DB9_2';
		arCalculateEnergy_1D[DB10_2].Name := 'DB10_2';
		arCalculateEnergy_1D[DB11_2].Name := 'DB11_2';
		arCalculateEnergy_1D[DB12_2].Name := 'DB12_2';
		arCalculateEnergy_1D[DB13_2].Name := 'DB13_2';
		arCalculateEnergy_1D[DB14_2].Name := 'DB14_2';
		arCalculateEnergy_1D[DB15_2].Name := 'DB15_2';
// set period time calculate
	// hour
		FOR iloop := 0 TO pmDev.numAllMeter - 1 DO
			arCalculateEnergy_1H[iloop].TimeAccumulate := NEW_HOUR;
		END_FOR
	// day
		FOR iloop := 0 TO pmDev.numAllMeter - 1 DO
			arCalculateEnergy_1D[iloop].TimeAccumulate := NEW_DAY;
		END_FOR
// Init calculate
		FOR iloop := 0 TO pmDev.numAllMeter - 1 DO
			arCalculateEnergy_1H[iloop].MR_Init();
		END_FOR
// Init Calculate Day
		FOR iloop := 0 TO pmDev.numAllMeter - 1 DO
			arCalculateEnergy_1D[iloop].MR_Init ();
		END_FOR
// check Init ok calculate
		FOR iloop := 0 TO pmDev.numAllMeter - 1 DO
			IF NOT arCalculateEnergy_1H[iloop].isRuning THEN
				AllInitSuccessful := FALSE;
			END_IF
		END_FOR
// check Init ok  Calculate Day
		FOR iloop := 0 TO pmDev.numAllMeter - 1 DO
			IF NOT arCalculateEnergy_1D[iloop].isRuning THEN
				AllInitSuccessful := FALSE;
			END_IF
		END_FOR
// 	change step
		IF AllInitSuccessful THEN
			eState := STATE_RUN;
		END_IF
END_METHOD

METHOD Run : BOOL
VAR_INPUT
END_VAR
VAR 
	iLoop : UINT;

